// TIA Portal V17 export
// export: Created 2025-03-05T08:01:40.8595336Z, ExportSetting WithDefaults, DisplayName Totally Integrated Automation Portal, DisplayVersion V17 Update 8, DisplayName TIA Portal Openness, DisplayVersion V17 Update 8, DisplayName TIA Portal Version Control Interface, DisplayVersion V17, DisplayName SINAMICS Startdrive Advanced, DisplayVersion V17 SP2, DisplayName SINAMICS Startdrive G110M, G120, G120C, G120D, G120P, G115D, DisplayVersion V17 SP2, DisplayName SINAMICS Startdrive G130, G150, S120, S150, SINAMICS MV, S210, DisplayVersion V17 SP2, DisplayName STEP 7 Professional, DisplayVersion V17 Update 8, DisplayName SINUMERIK ONE STEP 7 Toolbox, DisplayVersion V17 Update 12, DisplayName SINUMERIK 840D sl STEP 7 Toolbox, DisplayVersion V17 Update 12, DisplayName STEP 7 Safety, DisplayVersion V17 Update 6, DisplayName WinCC Advanced, DisplayVersion V17 Update 8
FUNCTION "FC7238_HMI_WINCC_OVERVIEW" : Void   // FC7238, LAD
{ S7_Optimized_Access := 'TRUE' }
VERSION : 0.1
// stored: AutoNumber false, IsIECCheckEnabled false, SetENOAutomatically false, UDAEnableTagReadback false
   VAR_TEMP
      RETVAL_FILL : Int;
   END_VAR
BEGIN

REGION Network 1: UNIT 01 ASPIRATION ALL STATIONS READY
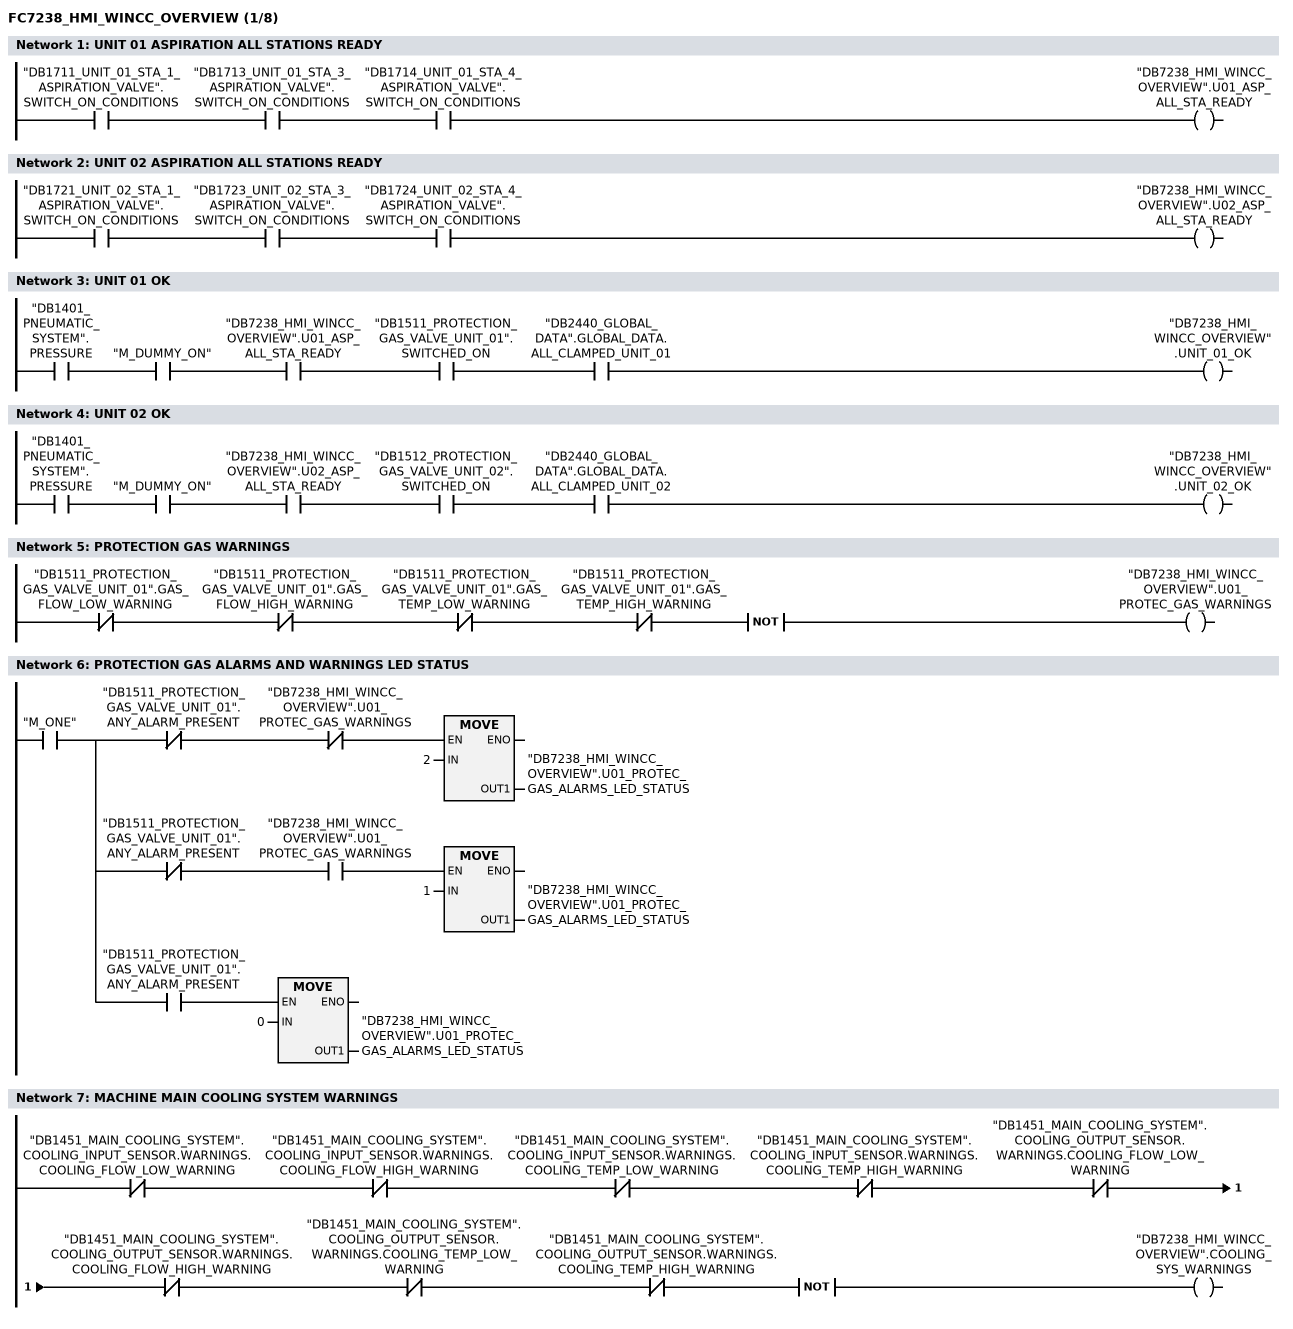
   RUNG wire#powerrail
      Contact( "DB1711_UNIT_01_STA_1_ASPIRATION_VALVE".SWITCH_ON_CONDITIONS )
      Contact( "DB1713_UNIT_01_STA_3_ASPIRATION_VALVE".SWITCH_ON_CONDITIONS )
      Contact( "DB1714_UNIT_01_STA_4_ASPIRATION_VALVE".SWITCH_ON_CONDITIONS )
      Coil( "DB7238_HMI_WINCC_OVERVIEW".U01_ASP_ALL_STA_READY )
   END_RUNG
   // the same network as SCL:
   "DB7238_HMI_WINCC_OVERVIEW".U01_ASP_ALL_STA_READY := "DB1711_UNIT_01_STA_1_ASPIRATION_VALVE".SWITCH_ON_CONDITIONS AND "DB1713_UNIT_01_STA_3_ASPIRATION_VALVE".SWITCH_ON_CONDITIONS AND "DB1714_UNIT_01_STA_4_ASPIRATION_VALVE".SWITCH_ON_CONDITIONS;
END_REGION

REGION Network 2: UNIT 02 ASPIRATION ALL STATIONS READY
   RUNG wire#powerrail
      Contact( "DB1721_UNIT_02_STA_1_ASPIRATION_VALVE".SWITCH_ON_CONDITIONS )
      Contact( "DB1723_UNIT_02_STA_3_ASPIRATION_VALVE".SWITCH_ON_CONDITIONS )
      Contact( "DB1724_UNIT_02_STA_4_ASPIRATION_VALVE".SWITCH_ON_CONDITIONS )
      Coil( "DB7238_HMI_WINCC_OVERVIEW".U02_ASP_ALL_STA_READY )
   END_RUNG
   // the same network as SCL:
   "DB7238_HMI_WINCC_OVERVIEW".U02_ASP_ALL_STA_READY := "DB1721_UNIT_02_STA_1_ASPIRATION_VALVE".SWITCH_ON_CONDITIONS AND "DB1723_UNIT_02_STA_3_ASPIRATION_VALVE".SWITCH_ON_CONDITIONS AND "DB1724_UNIT_02_STA_4_ASPIRATION_VALVE".SWITCH_ON_CONDITIONS;
END_REGION

REGION Network 3: UNIT 01 OK
   RUNG wire#powerrail
      Contact( "DB1401_PNEUMATIC_SYSTEM".PRESSURE )
      Contact( "M_DUMMY_ON" )
      Contact( "DB7238_HMI_WINCC_OVERVIEW".U01_ASP_ALL_STA_READY )
      Contact( "DB1511_PROTECTION_GAS_VALVE_UNIT_01".SWITCHED_ON )
      Contact( "DB2440_GLOBAL_DATA".GLOBAL_DATA.ALL_CLAMPED_UNIT_01 )
      Coil( "DB7238_HMI_WINCC_OVERVIEW".UNIT_01_OK )
   END_RUNG
   // the same network as SCL:
   "DB7238_HMI_WINCC_OVERVIEW".UNIT_01_OK := "DB1401_PNEUMATIC_SYSTEM".PRESSURE AND "M_DUMMY_ON" AND "DB7238_HMI_WINCC_OVERVIEW".U01_ASP_ALL_STA_READY AND "DB1511_PROTECTION_GAS_VALVE_UNIT_01".SWITCHED_ON AND "DB2440_GLOBAL_DATA".GLOBAL_DATA.ALL_CLAMPED_UNIT_01;
END_REGION

REGION Network 4: UNIT 02 OK
   RUNG wire#powerrail
      Contact( "DB1401_PNEUMATIC_SYSTEM".PRESSURE )
      Contact( "M_DUMMY_ON" )
      Contact( "DB7238_HMI_WINCC_OVERVIEW".U02_ASP_ALL_STA_READY )
      Contact( "DB1512_PROTECTION_GAS_VALVE_UNIT_02".SWITCHED_ON )
      Contact( "DB2440_GLOBAL_DATA".GLOBAL_DATA.ALL_CLAMPED_UNIT_02 )
      Coil( "DB7238_HMI_WINCC_OVERVIEW".UNIT_02_OK )
   END_RUNG
   // the same network as SCL:
   "DB7238_HMI_WINCC_OVERVIEW".UNIT_02_OK := "DB1401_PNEUMATIC_SYSTEM".PRESSURE AND "M_DUMMY_ON" AND "DB7238_HMI_WINCC_OVERVIEW".U02_ASP_ALL_STA_READY AND "DB1512_PROTECTION_GAS_VALVE_UNIT_02".SWITCHED_ON AND "DB2440_GLOBAL_DATA".GLOBAL_DATA.ALL_CLAMPED_UNIT_02;
END_REGION

REGION Network 5: PROTECTION GAS WARNINGS
   RUNG wire#powerrail
      I_Contact( "DB1511_PROTECTION_GAS_VALVE_UNIT_01".GAS_FLOW_LOW_WARNING )
      I_Contact( "DB1511_PROTECTION_GAS_VALVE_UNIT_01".GAS_FLOW_HIGH_WARNING )
      I_Contact( "DB1511_PROTECTION_GAS_VALVE_UNIT_01".GAS_TEMP_LOW_WARNING )
      I_Contact( "DB1511_PROTECTION_GAS_VALVE_UNIT_01".GAS_TEMP_HIGH_WARNING )
      Not()
      Coil( "DB7238_HMI_WINCC_OVERVIEW".U01_PROTEC_GAS_WARNINGS )
   END_RUNG
   // the same network as SCL:
   "DB7238_HMI_WINCC_OVERVIEW".U01_PROTEC_GAS_WARNINGS := NOT (NOT "DB1511_PROTECTION_GAS_VALVE_UNIT_01".GAS_FLOW_LOW_WARNING AND NOT "DB1511_PROTECTION_GAS_VALVE_UNIT_01".GAS_FLOW_HIGH_WARNING AND NOT "DB1511_PROTECTION_GAS_VALVE_UNIT_01".GAS_TEMP_LOW_WARNING AND NOT "DB1511_PROTECTION_GAS_VALVE_UNIT_01".GAS_TEMP_HIGH_WARNING);
END_REGION

REGION Network 6: PROTECTION GAS ALARMS AND WARNINGS LED STATUS
   RUNG wire#powerrail
      Contact( "M_ONE" )
      wire#w1
      I_Contact( "DB1511_PROTECTION_GAS_VALVE_UNIT_01".ANY_ALARM_PRESENT )
      I_Contact( "DB7238_HMI_WINCC_OVERVIEW".U01_PROTEC_GAS_WARNINGS )
      { S7_GenerateENO := "TRUE" } Move(in := 2, out1 => "DB7238_HMI_WINCC_OVERVIEW".U01_PROTEC_GAS_ALARMS_LED_STATUS)
   END_RUNG
   RUNG wire#w1
      I_Contact( "DB1511_PROTECTION_GAS_VALVE_UNIT_01".ANY_ALARM_PRESENT )
      Contact( "DB7238_HMI_WINCC_OVERVIEW".U01_PROTEC_GAS_WARNINGS )
      { S7_GenerateENO := "TRUE" } Move(in := 1, out1 => "DB7238_HMI_WINCC_OVERVIEW".U01_PROTEC_GAS_ALARMS_LED_STATUS)
   END_RUNG
   RUNG wire#w1
      Contact( "DB1511_PROTECTION_GAS_VALVE_UNIT_01".ANY_ALARM_PRESENT )
      { S7_GenerateENO := "TRUE" } Move(in := 0, out1 => "DB7238_HMI_WINCC_OVERVIEW".U01_PROTEC_GAS_ALARMS_LED_STATUS)
   END_RUNG
   // the same network as SCL:
   IF "M_ONE" AND NOT "DB1511_PROTECTION_GAS_VALVE_UNIT_01".ANY_ALARM_PRESENT AND NOT "DB7238_HMI_WINCC_OVERVIEW".U01_PROTEC_GAS_WARNINGS THEN
       "DB7238_HMI_WINCC_OVERVIEW".U01_PROTEC_GAS_ALARMS_LED_STATUS := 2;
   END_IF;
   IF "M_ONE" AND NOT "DB1511_PROTECTION_GAS_VALVE_UNIT_01".ANY_ALARM_PRESENT AND "DB7238_HMI_WINCC_OVERVIEW".U01_PROTEC_GAS_WARNINGS THEN
       "DB7238_HMI_WINCC_OVERVIEW".U01_PROTEC_GAS_ALARMS_LED_STATUS := 1;
   END_IF;
   IF "M_ONE" AND "DB1511_PROTECTION_GAS_VALVE_UNIT_01".ANY_ALARM_PRESENT THEN
       "DB7238_HMI_WINCC_OVERVIEW".U01_PROTEC_GAS_ALARMS_LED_STATUS := 0;
   END_IF;
END_REGION

REGION Network 7: MACHINE MAIN COOLING SYSTEM WARNINGS
   RUNG wire#powerrail
      I_Contact( "DB1451_MAIN_COOLING_SYSTEM".COOLING_INPUT_SENSOR.WARNINGS.COOLING_FLOW_LOW_WARNING )
      I_Contact( "DB1451_MAIN_COOLING_SYSTEM".COOLING_INPUT_SENSOR.WARNINGS.COOLING_FLOW_HIGH_WARNING )
      I_Contact( "DB1451_MAIN_COOLING_SYSTEM".COOLING_INPUT_SENSOR.WARNINGS.COOLING_TEMP_LOW_WARNING )
      I_Contact( "DB1451_MAIN_COOLING_SYSTEM".COOLING_INPUT_SENSOR.WARNINGS.COOLING_TEMP_HIGH_WARNING )
      I_Contact( "DB1451_MAIN_COOLING_SYSTEM".COOLING_OUTPUT_SENSOR.WARNINGS.COOLING_FLOW_LOW_WARNING )
      I_Contact( "DB1451_MAIN_COOLING_SYSTEM".COOLING_OUTPUT_SENSOR.WARNINGS.COOLING_FLOW_HIGH_WARNING )
      I_Contact( "DB1451_MAIN_COOLING_SYSTEM".COOLING_OUTPUT_SENSOR.WARNINGS.COOLING_TEMP_LOW_WARNING )
      I_Contact( "DB1451_MAIN_COOLING_SYSTEM".COOLING_OUTPUT_SENSOR.WARNINGS.COOLING_TEMP_HIGH_WARNING )
      Not()
      Coil( "DB7238_HMI_WINCC_OVERVIEW".COOLING_SYS_WARNINGS )
   END_RUNG
   // the same network as SCL:
   "DB7238_HMI_WINCC_OVERVIEW".COOLING_SYS_WARNINGS := NOT (NOT "DB1451_MAIN_COOLING_SYSTEM".COOLING_INPUT_SENSOR.WARNINGS.COOLING_FLOW_LOW_WARNING AND NOT "DB1451_MAIN_COOLING_SYSTEM".COOLING_INPUT_SENSOR.WARNINGS.COOLING_FLOW_HIGH_WARNING AND NOT "DB1451_MAIN_COOLING_SYSTEM".COOLING_INPUT_SENSOR.WARNINGS.COOLING_TEMP_LOW_WARNING AND NOT "DB1451_MAIN_COOLING_SYSTEM".COOLING_INPUT_SENSOR.WARNINGS.COOLING_TEMP_HIGH_WARNING AND NOT "DB1451_MAIN_COOLING_SYSTEM".COOLING_OUTPUT_SENSOR.WARNINGS.COOLING_FLOW_LOW_WARNING AND NOT "DB1451_MAIN_COOLING_SYSTEM".COOLING_OUTPUT_SENSOR.WARNINGS.COOLING_FLOW_HIGH_WARNING AND NOT "DB1451_MAIN_COOLING_SYSTEM".COOLING_OUTPUT_SENSOR.WARNINGS.COOLING_TEMP_LOW_WARNING AND NOT "DB1451_MAIN_COOLING_SYSTEM".COOLING_OUTPUT_SENSOR.WARNINGS.COOLING_TEMP_HIGH_WARNING);
END_REGION

REGION Network 8: MACHINE MAIN COOLING SYSTEM ALARMS
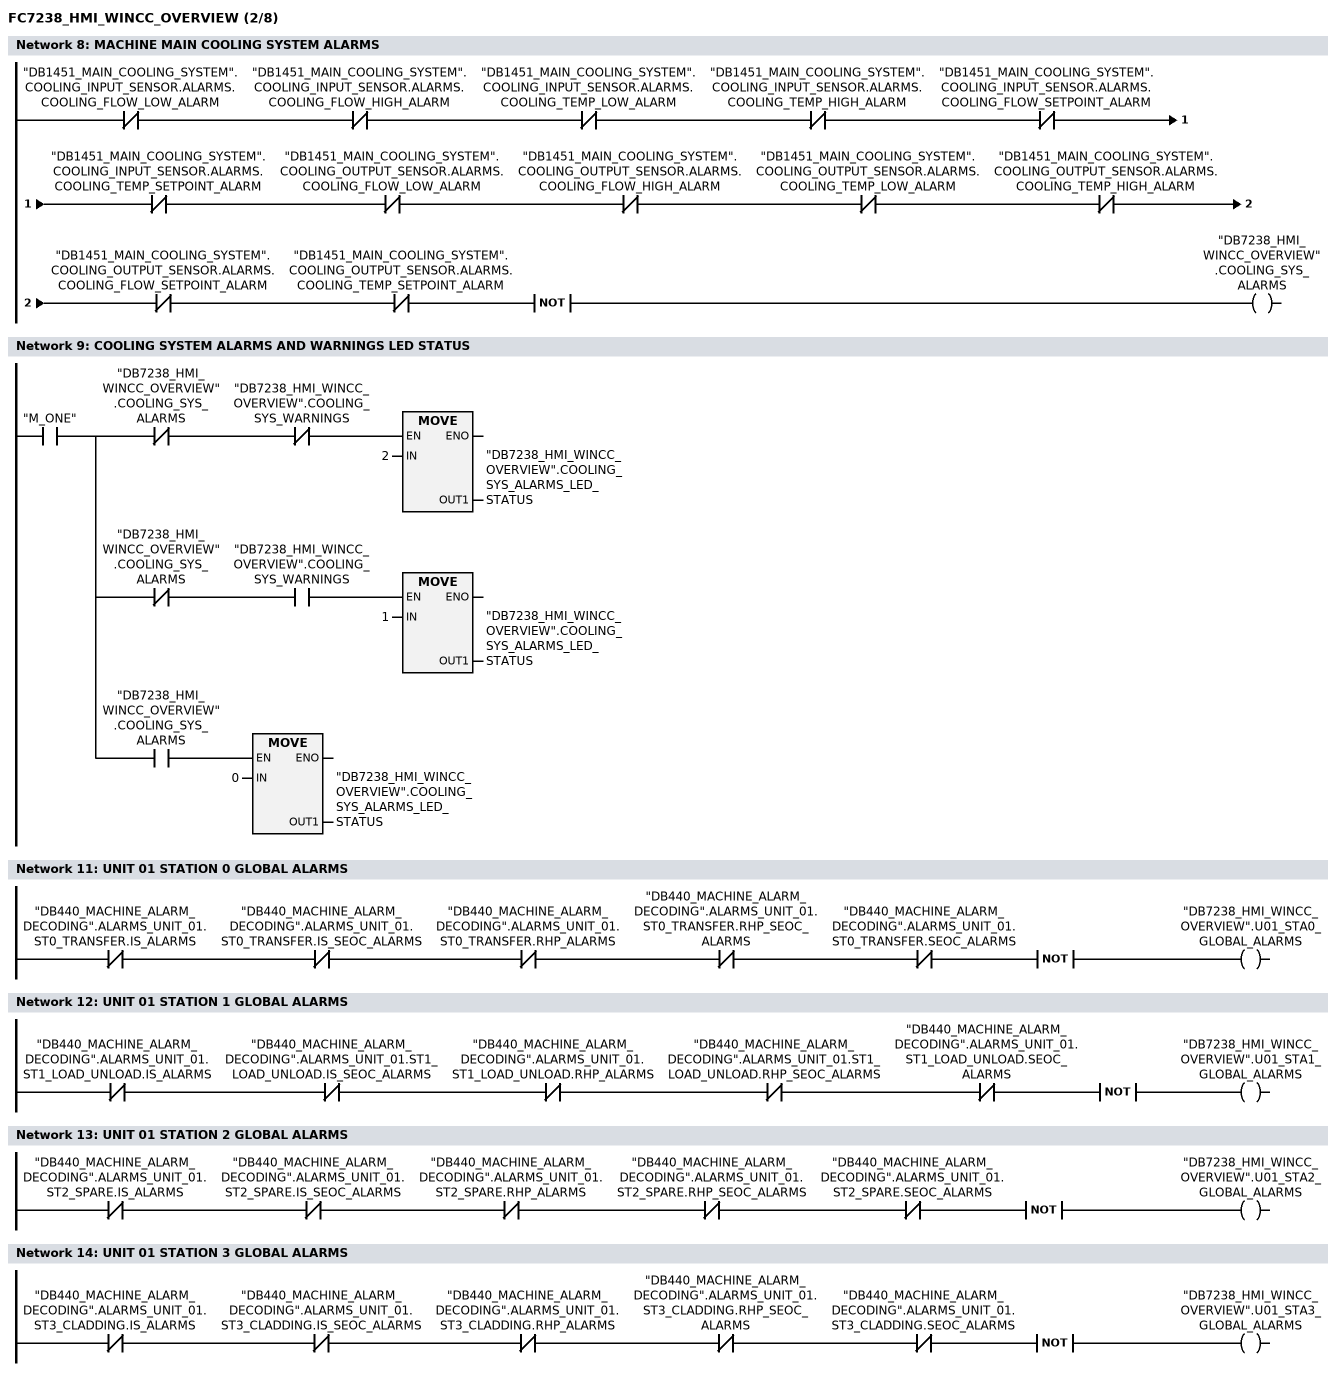
   RUNG wire#powerrail
      I_Contact( "DB1451_MAIN_COOLING_SYSTEM".COOLING_INPUT_SENSOR.ALARMS.COOLING_FLOW_LOW_ALARM )
      I_Contact( "DB1451_MAIN_COOLING_SYSTEM".COOLING_INPUT_SENSOR.ALARMS.COOLING_FLOW_HIGH_ALARM )
      I_Contact( "DB1451_MAIN_COOLING_SYSTEM".COOLING_INPUT_SENSOR.ALARMS.COOLING_TEMP_LOW_ALARM )
      I_Contact( "DB1451_MAIN_COOLING_SYSTEM".COOLING_INPUT_SENSOR.ALARMS.COOLING_TEMP_HIGH_ALARM )
      I_Contact( "DB1451_MAIN_COOLING_SYSTEM".COOLING_INPUT_SENSOR.ALARMS.COOLING_FLOW_SETPOINT_ALARM )
      I_Contact( "DB1451_MAIN_COOLING_SYSTEM".COOLING_INPUT_SENSOR.ALARMS.COOLING_TEMP_SETPOINT_ALARM )
      I_Contact( "DB1451_MAIN_COOLING_SYSTEM".COOLING_OUTPUT_SENSOR.ALARMS.COOLING_FLOW_LOW_ALARM )
      I_Contact( "DB1451_MAIN_COOLING_SYSTEM".COOLING_OUTPUT_SENSOR.ALARMS.COOLING_FLOW_HIGH_ALARM )
      I_Contact( "DB1451_MAIN_COOLING_SYSTEM".COOLING_OUTPUT_SENSOR.ALARMS.COOLING_TEMP_LOW_ALARM )
      I_Contact( "DB1451_MAIN_COOLING_SYSTEM".COOLING_OUTPUT_SENSOR.ALARMS.COOLING_TEMP_HIGH_ALARM )
      I_Contact( "DB1451_MAIN_COOLING_SYSTEM".COOLING_OUTPUT_SENSOR.ALARMS.COOLING_FLOW_SETPOINT_ALARM )
      I_Contact( "DB1451_MAIN_COOLING_SYSTEM".COOLING_OUTPUT_SENSOR.ALARMS.COOLING_TEMP_SETPOINT_ALARM )
      Not()
      Coil( "DB7238_HMI_WINCC_OVERVIEW".COOLING_SYS_ALARMS )
   END_RUNG
   // the same network as SCL:
   "DB7238_HMI_WINCC_OVERVIEW".COOLING_SYS_ALARMS := NOT (NOT "DB1451_MAIN_COOLING_SYSTEM".COOLING_INPUT_SENSOR.ALARMS.COOLING_FLOW_LOW_ALARM AND NOT "DB1451_MAIN_COOLING_SYSTEM".COOLING_INPUT_SENSOR.ALARMS.COOLING_FLOW_HIGH_ALARM AND NOT "DB1451_MAIN_COOLING_SYSTEM".COOLING_INPUT_SENSOR.ALARMS.COOLING_TEMP_LOW_ALARM AND NOT "DB1451_MAIN_COOLING_SYSTEM".COOLING_INPUT_SENSOR.ALARMS.COOLING_TEMP_HIGH_ALARM AND NOT "DB1451_MAIN_COOLING_SYSTEM".COOLING_INPUT_SENSOR.ALARMS.COOLING_FLOW_SETPOINT_ALARM AND NOT "DB1451_MAIN_COOLING_SYSTEM".COOLING_INPUT_SENSOR.ALARMS.COOLING_TEMP_SETPOINT_ALARM AND NOT "DB1451_MAIN_COOLING_SYSTEM".COOLING_OUTPUT_SENSOR.ALARMS.COOLING_FLOW_LOW_ALARM AND NOT "DB1451_MAIN_COOLING_SYSTEM".COOLING_OUTPUT_SENSOR.ALARMS.COOLING_FLOW_HIGH_ALARM AND NOT "DB1451_MAIN_COOLING_SYSTEM".COOLING_OUTPUT_SENSOR.ALARMS.COOLING_TEMP_LOW_ALARM AND NOT "DB1451_MAIN_COOLING_SYSTEM".COOLING_OUTPUT_SENSOR.ALARMS.COOLING_TEMP_HIGH_ALARM AND NOT "DB1451_MAIN_COOLING_SYSTEM".COOLING_OUTPUT_SENSOR.ALARMS.COOLING_FLOW_SETPOINT_ALARM AND NOT "DB1451_MAIN_COOLING_SYSTEM".COOLING_OUTPUT_SENSOR.ALARMS.COOLING_TEMP_SETPOINT_ALARM);
END_REGION

REGION Network 9: COOLING SYSTEM ALARMS AND WARNINGS LED STATUS
   RUNG wire#powerrail
      Contact( "M_ONE" )
      wire#w1
      I_Contact( "DB7238_HMI_WINCC_OVERVIEW".COOLING_SYS_ALARMS )
      I_Contact( "DB7238_HMI_WINCC_OVERVIEW".COOLING_SYS_WARNINGS )
      { S7_GenerateENO := "TRUE" } Move(in := 2, out1 => "DB7238_HMI_WINCC_OVERVIEW".COOLING_SYS_ALARMS_LED_STATUS)
   END_RUNG
   RUNG wire#w1
      I_Contact( "DB7238_HMI_WINCC_OVERVIEW".COOLING_SYS_ALARMS )
      Contact( "DB7238_HMI_WINCC_OVERVIEW".COOLING_SYS_WARNINGS )
      { S7_GenerateENO := "TRUE" } Move(in := 1, out1 => "DB7238_HMI_WINCC_OVERVIEW".COOLING_SYS_ALARMS_LED_STATUS)
   END_RUNG
   RUNG wire#w1
      Contact( "DB7238_HMI_WINCC_OVERVIEW".COOLING_SYS_ALARMS )
      { S7_GenerateENO := "TRUE" } Move(in := 0, out1 => "DB7238_HMI_WINCC_OVERVIEW".COOLING_SYS_ALARMS_LED_STATUS)
   END_RUNG
   // the same network as SCL:
   IF "M_ONE" AND NOT "DB7238_HMI_WINCC_OVERVIEW".COOLING_SYS_ALARMS AND NOT "DB7238_HMI_WINCC_OVERVIEW".COOLING_SYS_WARNINGS THEN
       "DB7238_HMI_WINCC_OVERVIEW".COOLING_SYS_ALARMS_LED_STATUS := 2;
   END_IF;
   IF "M_ONE" AND NOT "DB7238_HMI_WINCC_OVERVIEW".COOLING_SYS_ALARMS AND "DB7238_HMI_WINCC_OVERVIEW".COOLING_SYS_WARNINGS THEN
       "DB7238_HMI_WINCC_OVERVIEW".COOLING_SYS_ALARMS_LED_STATUS := 1;
   END_IF;
   IF "M_ONE" AND "DB7238_HMI_WINCC_OVERVIEW".COOLING_SYS_ALARMS THEN
       "DB7238_HMI_WINCC_OVERVIEW".COOLING_SYS_ALARMS_LED_STATUS := 0;
   END_IF;
END_REGION

REGION Network 10: <<<<<<<<<<<<<<<<<<<<<<<< UNIT 01 >>>>>>>>>>>>>>>>>>>>>>>>
END_REGION

REGION Network 11: UNIT 01 STATION 0 GLOBAL ALARMS
   RUNG wire#powerrail
      I_Contact( "DB440_MACHINE_ALARM_DECODING".ALARMS_UNIT_01.ST0_TRANSFER.IS_ALARMS )
      I_Contact( "DB440_MACHINE_ALARM_DECODING".ALARMS_UNIT_01.ST0_TRANSFER.IS_SEOC_ALARMS )
      I_Contact( "DB440_MACHINE_ALARM_DECODING".ALARMS_UNIT_01.ST0_TRANSFER.RHP_ALARMS )
      I_Contact( "DB440_MACHINE_ALARM_DECODING".ALARMS_UNIT_01.ST0_TRANSFER.RHP_SEOC_ALARMS )
      I_Contact( "DB440_MACHINE_ALARM_DECODING".ALARMS_UNIT_01.ST0_TRANSFER.SEOC_ALARMS )
      Not()
      Coil( "DB7238_HMI_WINCC_OVERVIEW".U01_STA0_GLOBAL_ALARMS )
   END_RUNG
   // the same network as SCL:
   "DB7238_HMI_WINCC_OVERVIEW".U01_STA0_GLOBAL_ALARMS := NOT (NOT "DB440_MACHINE_ALARM_DECODING".ALARMS_UNIT_01.ST0_TRANSFER.IS_ALARMS AND NOT "DB440_MACHINE_ALARM_DECODING".ALARMS_UNIT_01.ST0_TRANSFER.IS_SEOC_ALARMS AND NOT "DB440_MACHINE_ALARM_DECODING".ALARMS_UNIT_01.ST0_TRANSFER.RHP_ALARMS AND NOT "DB440_MACHINE_ALARM_DECODING".ALARMS_UNIT_01.ST0_TRANSFER.RHP_SEOC_ALARMS AND NOT "DB440_MACHINE_ALARM_DECODING".ALARMS_UNIT_01.ST0_TRANSFER.SEOC_ALARMS);
END_REGION

REGION Network 12: UNIT 01 STATION 1 GLOBAL ALARMS
   RUNG wire#powerrail
      I_Contact( "DB440_MACHINE_ALARM_DECODING".ALARMS_UNIT_01.ST1_LOAD_UNLOAD.IS_ALARMS )
      I_Contact( "DB440_MACHINE_ALARM_DECODING".ALARMS_UNIT_01.ST1_LOAD_UNLOAD.IS_SEOC_ALARMS )
      I_Contact( "DB440_MACHINE_ALARM_DECODING".ALARMS_UNIT_01.ST1_LOAD_UNLOAD.RHP_ALARMS )
      I_Contact( "DB440_MACHINE_ALARM_DECODING".ALARMS_UNIT_01.ST1_LOAD_UNLOAD.RHP_SEOC_ALARMS )
      I_Contact( "DB440_MACHINE_ALARM_DECODING".ALARMS_UNIT_01.ST1_LOAD_UNLOAD.SEOC_ALARMS )
      Not()
      Coil( "DB7238_HMI_WINCC_OVERVIEW".U01_STA1_GLOBAL_ALARMS )
   END_RUNG
   // the same network as SCL:
   "DB7238_HMI_WINCC_OVERVIEW".U01_STA1_GLOBAL_ALARMS := NOT (NOT "DB440_MACHINE_ALARM_DECODING".ALARMS_UNIT_01.ST1_LOAD_UNLOAD.IS_ALARMS AND NOT "DB440_MACHINE_ALARM_DECODING".ALARMS_UNIT_01.ST1_LOAD_UNLOAD.IS_SEOC_ALARMS AND NOT "DB440_MACHINE_ALARM_DECODING".ALARMS_UNIT_01.ST1_LOAD_UNLOAD.RHP_ALARMS AND NOT "DB440_MACHINE_ALARM_DECODING".ALARMS_UNIT_01.ST1_LOAD_UNLOAD.RHP_SEOC_ALARMS AND NOT "DB440_MACHINE_ALARM_DECODING".ALARMS_UNIT_01.ST1_LOAD_UNLOAD.SEOC_ALARMS);
END_REGION

REGION Network 13: UNIT 01 STATION 2 GLOBAL ALARMS
   RUNG wire#powerrail
      I_Contact( "DB440_MACHINE_ALARM_DECODING".ALARMS_UNIT_01.ST2_SPARE.IS_ALARMS )
      I_Contact( "DB440_MACHINE_ALARM_DECODING".ALARMS_UNIT_01.ST2_SPARE.IS_SEOC_ALARMS )
      I_Contact( "DB440_MACHINE_ALARM_DECODING".ALARMS_UNIT_01.ST2_SPARE.RHP_ALARMS )
      I_Contact( "DB440_MACHINE_ALARM_DECODING".ALARMS_UNIT_01.ST2_SPARE.RHP_SEOC_ALARMS )
      I_Contact( "DB440_MACHINE_ALARM_DECODING".ALARMS_UNIT_01.ST2_SPARE.SEOC_ALARMS )
      Not()
      Coil( "DB7238_HMI_WINCC_OVERVIEW".U01_STA2_GLOBAL_ALARMS )
   END_RUNG
   // the same network as SCL:
   "DB7238_HMI_WINCC_OVERVIEW".U01_STA2_GLOBAL_ALARMS := NOT (NOT "DB440_MACHINE_ALARM_DECODING".ALARMS_UNIT_01.ST2_SPARE.IS_ALARMS AND NOT "DB440_MACHINE_ALARM_DECODING".ALARMS_UNIT_01.ST2_SPARE.IS_SEOC_ALARMS AND NOT "DB440_MACHINE_ALARM_DECODING".ALARMS_UNIT_01.ST2_SPARE.RHP_ALARMS AND NOT "DB440_MACHINE_ALARM_DECODING".ALARMS_UNIT_01.ST2_SPARE.RHP_SEOC_ALARMS AND NOT "DB440_MACHINE_ALARM_DECODING".ALARMS_UNIT_01.ST2_SPARE.SEOC_ALARMS);
END_REGION

REGION Network 14: UNIT 01 STATION 3 GLOBAL ALARMS
   RUNG wire#powerrail
      I_Contact( "DB440_MACHINE_ALARM_DECODING".ALARMS_UNIT_01.ST3_CLADDING.IS_ALARMS )
      I_Contact( "DB440_MACHINE_ALARM_DECODING".ALARMS_UNIT_01.ST3_CLADDING.IS_SEOC_ALARMS )
      I_Contact( "DB440_MACHINE_ALARM_DECODING".ALARMS_UNIT_01.ST3_CLADDING.RHP_ALARMS )
      I_Contact( "DB440_MACHINE_ALARM_DECODING".ALARMS_UNIT_01.ST3_CLADDING.RHP_SEOC_ALARMS )
      I_Contact( "DB440_MACHINE_ALARM_DECODING".ALARMS_UNIT_01.ST3_CLADDING.SEOC_ALARMS )
      Not()
      Coil( "DB7238_HMI_WINCC_OVERVIEW".U01_STA3_GLOBAL_ALARMS )
   END_RUNG
   // the same network as SCL:
   "DB7238_HMI_WINCC_OVERVIEW".U01_STA3_GLOBAL_ALARMS := NOT (NOT "DB440_MACHINE_ALARM_DECODING".ALARMS_UNIT_01.ST3_CLADDING.IS_ALARMS AND NOT "DB440_MACHINE_ALARM_DECODING".ALARMS_UNIT_01.ST3_CLADDING.IS_SEOC_ALARMS AND NOT "DB440_MACHINE_ALARM_DECODING".ALARMS_UNIT_01.ST3_CLADDING.RHP_ALARMS AND NOT "DB440_MACHINE_ALARM_DECODING".ALARMS_UNIT_01.ST3_CLADDING.RHP_SEOC_ALARMS AND NOT "DB440_MACHINE_ALARM_DECODING".ALARMS_UNIT_01.ST3_CLADDING.SEOC_ALARMS);
END_REGION

REGION Network 15: UNIT 01 STATION 4 GLOBAL ALARMS
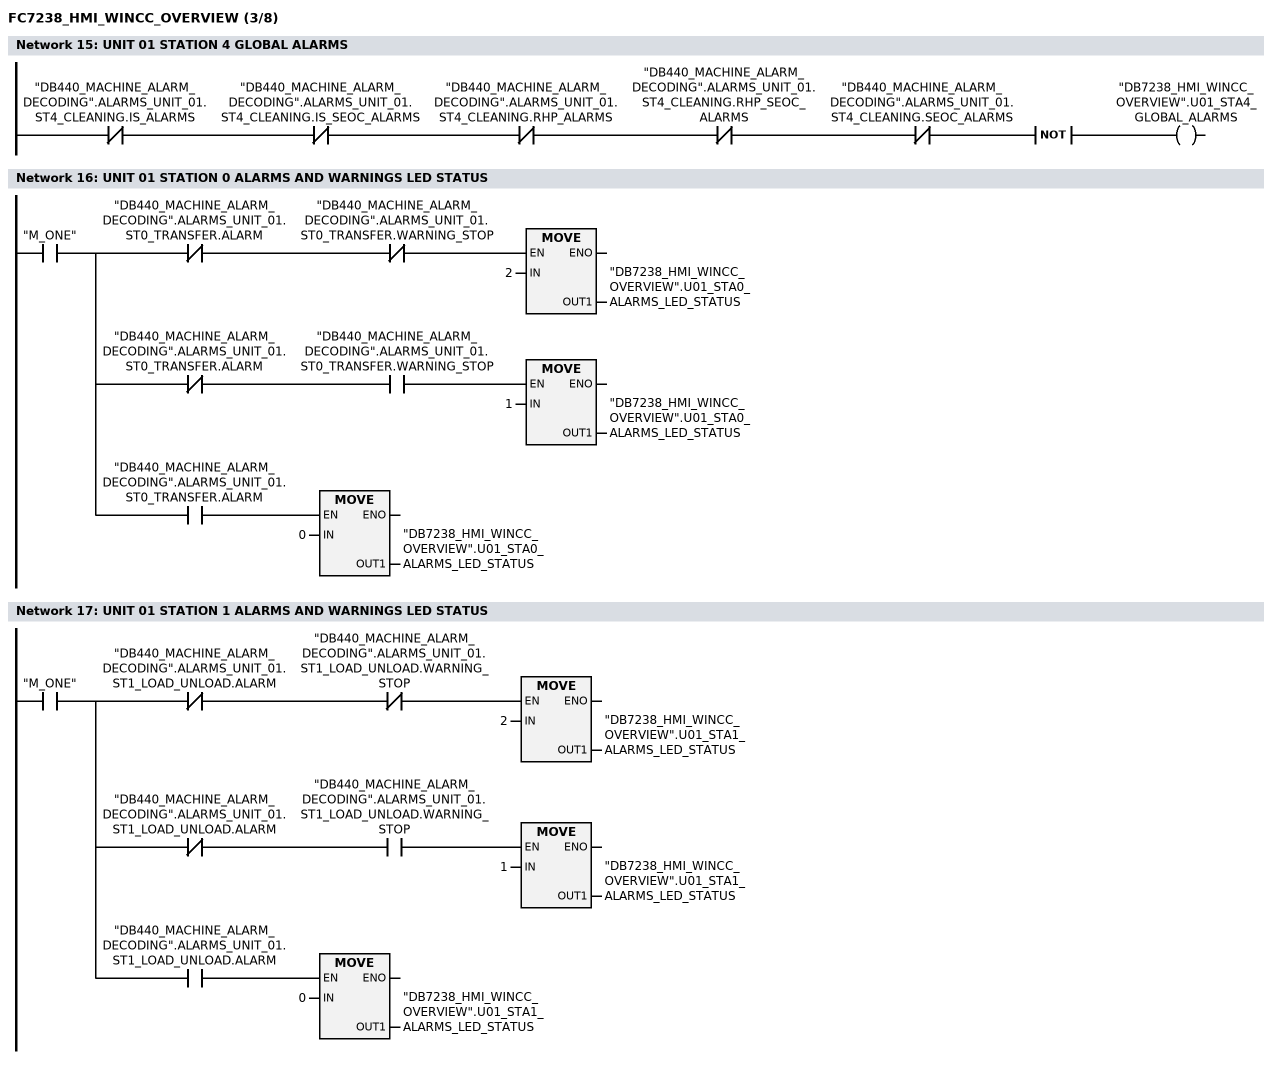
   RUNG wire#powerrail
      I_Contact( "DB440_MACHINE_ALARM_DECODING".ALARMS_UNIT_01.ST4_CLEANING.IS_ALARMS )
      I_Contact( "DB440_MACHINE_ALARM_DECODING".ALARMS_UNIT_01.ST4_CLEANING.IS_SEOC_ALARMS )
      I_Contact( "DB440_MACHINE_ALARM_DECODING".ALARMS_UNIT_01.ST4_CLEANING.RHP_ALARMS )
      I_Contact( "DB440_MACHINE_ALARM_DECODING".ALARMS_UNIT_01.ST4_CLEANING.RHP_SEOC_ALARMS )
      I_Contact( "DB440_MACHINE_ALARM_DECODING".ALARMS_UNIT_01.ST4_CLEANING.SEOC_ALARMS )
      Not()
      Coil( "DB7238_HMI_WINCC_OVERVIEW".U01_STA4_GLOBAL_ALARMS )
   END_RUNG
   // the same network as SCL:
   "DB7238_HMI_WINCC_OVERVIEW".U01_STA4_GLOBAL_ALARMS := NOT (NOT "DB440_MACHINE_ALARM_DECODING".ALARMS_UNIT_01.ST4_CLEANING.IS_ALARMS AND NOT "DB440_MACHINE_ALARM_DECODING".ALARMS_UNIT_01.ST4_CLEANING.IS_SEOC_ALARMS AND NOT "DB440_MACHINE_ALARM_DECODING".ALARMS_UNIT_01.ST4_CLEANING.RHP_ALARMS AND NOT "DB440_MACHINE_ALARM_DECODING".ALARMS_UNIT_01.ST4_CLEANING.RHP_SEOC_ALARMS AND NOT "DB440_MACHINE_ALARM_DECODING".ALARMS_UNIT_01.ST4_CLEANING.SEOC_ALARMS);
END_REGION

REGION Network 16: UNIT 01 STATION 0 ALARMS AND WARNINGS LED STATUS
   RUNG wire#powerrail
      Contact( "M_ONE" )
      wire#w1
      I_Contact( "DB440_MACHINE_ALARM_DECODING".ALARMS_UNIT_01.ST0_TRANSFER.ALARM )
      I_Contact( "DB440_MACHINE_ALARM_DECODING".ALARMS_UNIT_01.ST0_TRANSFER.WARNING_STOP )
      { S7_GenerateENO := "TRUE" } Move(in := 2, out1 => "DB7238_HMI_WINCC_OVERVIEW".U01_STA0_ALARMS_LED_STATUS)
   END_RUNG
   RUNG wire#w1
      I_Contact( "DB440_MACHINE_ALARM_DECODING".ALARMS_UNIT_01.ST0_TRANSFER.ALARM )
      Contact( "DB440_MACHINE_ALARM_DECODING".ALARMS_UNIT_01.ST0_TRANSFER.WARNING_STOP )
      { S7_GenerateENO := "TRUE" } Move(in := 1, out1 => "DB7238_HMI_WINCC_OVERVIEW".U01_STA0_ALARMS_LED_STATUS)
   END_RUNG
   RUNG wire#w1
      Contact( "DB440_MACHINE_ALARM_DECODING".ALARMS_UNIT_01.ST0_TRANSFER.ALARM )
      { S7_GenerateENO := "TRUE" } Move(in := 0, out1 => "DB7238_HMI_WINCC_OVERVIEW".U01_STA0_ALARMS_LED_STATUS)
   END_RUNG
   // the same network as SCL:
   IF "M_ONE" AND NOT "DB440_MACHINE_ALARM_DECODING".ALARMS_UNIT_01.ST0_TRANSFER.ALARM AND NOT "DB440_MACHINE_ALARM_DECODING".ALARMS_UNIT_01.ST0_TRANSFER.WARNING_STOP THEN
       "DB7238_HMI_WINCC_OVERVIEW".U01_STA0_ALARMS_LED_STATUS := 2;
   END_IF;
   IF "M_ONE" AND NOT "DB440_MACHINE_ALARM_DECODING".ALARMS_UNIT_01.ST0_TRANSFER.ALARM AND "DB440_MACHINE_ALARM_DECODING".ALARMS_UNIT_01.ST0_TRANSFER.WARNING_STOP THEN
       "DB7238_HMI_WINCC_OVERVIEW".U01_STA0_ALARMS_LED_STATUS := 1;
   END_IF;
   IF "M_ONE" AND "DB440_MACHINE_ALARM_DECODING".ALARMS_UNIT_01.ST0_TRANSFER.ALARM THEN
       "DB7238_HMI_WINCC_OVERVIEW".U01_STA0_ALARMS_LED_STATUS := 0;
   END_IF;
END_REGION

REGION Network 17: UNIT 01 STATION 1 ALARMS AND WARNINGS LED STATUS
   RUNG wire#powerrail
      Contact( "M_ONE" )
      wire#w1
      I_Contact( "DB440_MACHINE_ALARM_DECODING".ALARMS_UNIT_01.ST1_LOAD_UNLOAD.ALARM )
      I_Contact( "DB440_MACHINE_ALARM_DECODING".ALARMS_UNIT_01.ST1_LOAD_UNLOAD.WARNING_STOP )
      { S7_GenerateENO := "TRUE" } Move(in := 2, out1 => "DB7238_HMI_WINCC_OVERVIEW".U01_STA1_ALARMS_LED_STATUS)
   END_RUNG
   RUNG wire#w1
      I_Contact( "DB440_MACHINE_ALARM_DECODING".ALARMS_UNIT_01.ST1_LOAD_UNLOAD.ALARM )
      Contact( "DB440_MACHINE_ALARM_DECODING".ALARMS_UNIT_01.ST1_LOAD_UNLOAD.WARNING_STOP )
      { S7_GenerateENO := "TRUE" } Move(in := 1, out1 => "DB7238_HMI_WINCC_OVERVIEW".U01_STA1_ALARMS_LED_STATUS)
   END_RUNG
   RUNG wire#w1
      Contact( "DB440_MACHINE_ALARM_DECODING".ALARMS_UNIT_01.ST1_LOAD_UNLOAD.ALARM )
      { S7_GenerateENO := "TRUE" } Move(in := 0, out1 => "DB7238_HMI_WINCC_OVERVIEW".U01_STA1_ALARMS_LED_STATUS)
   END_RUNG
   // the same network as SCL:
   IF "M_ONE" AND NOT "DB440_MACHINE_ALARM_DECODING".ALARMS_UNIT_01.ST1_LOAD_UNLOAD.ALARM AND NOT "DB440_MACHINE_ALARM_DECODING".ALARMS_UNIT_01.ST1_LOAD_UNLOAD.WARNING_STOP THEN
       "DB7238_HMI_WINCC_OVERVIEW".U01_STA1_ALARMS_LED_STATUS := 2;
   END_IF;
   IF "M_ONE" AND NOT "DB440_MACHINE_ALARM_DECODING".ALARMS_UNIT_01.ST1_LOAD_UNLOAD.ALARM AND "DB440_MACHINE_ALARM_DECODING".ALARMS_UNIT_01.ST1_LOAD_UNLOAD.WARNING_STOP THEN
       "DB7238_HMI_WINCC_OVERVIEW".U01_STA1_ALARMS_LED_STATUS := 1;
   END_IF;
   IF "M_ONE" AND "DB440_MACHINE_ALARM_DECODING".ALARMS_UNIT_01.ST1_LOAD_UNLOAD.ALARM THEN
       "DB7238_HMI_WINCC_OVERVIEW".U01_STA1_ALARMS_LED_STATUS := 0;
   END_IF;
END_REGION

REGION Network 18: UNIT 01 STATION 2 ALARMS AND WARNINGS LED STATUS
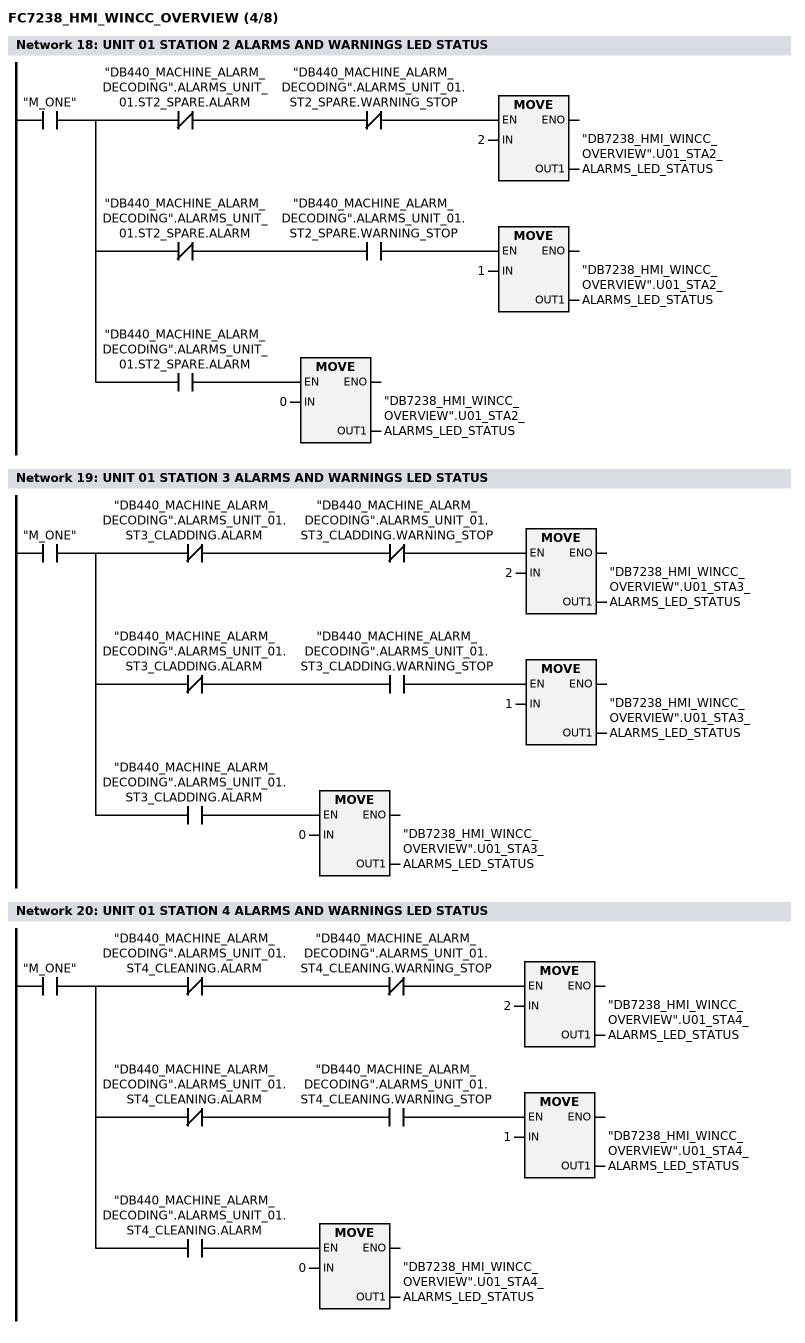
   RUNG wire#powerrail
      Contact( "M_ONE" )
      wire#w1
      I_Contact( "DB440_MACHINE_ALARM_DECODING".ALARMS_UNIT_01.ST2_SPARE.ALARM )
      I_Contact( "DB440_MACHINE_ALARM_DECODING".ALARMS_UNIT_01.ST2_SPARE.WARNING_STOP )
      { S7_GenerateENO := "TRUE" } Move(in := 2, out1 => "DB7238_HMI_WINCC_OVERVIEW".U01_STA2_ALARMS_LED_STATUS)
   END_RUNG
   RUNG wire#w1
      I_Contact( "DB440_MACHINE_ALARM_DECODING".ALARMS_UNIT_01.ST2_SPARE.ALARM )
      Contact( "DB440_MACHINE_ALARM_DECODING".ALARMS_UNIT_01.ST2_SPARE.WARNING_STOP )
      { S7_GenerateENO := "TRUE" } Move(in := 1, out1 => "DB7238_HMI_WINCC_OVERVIEW".U01_STA2_ALARMS_LED_STATUS)
   END_RUNG
   RUNG wire#w1
      Contact( "DB440_MACHINE_ALARM_DECODING".ALARMS_UNIT_01.ST2_SPARE.ALARM )
      { S7_GenerateENO := "TRUE" } Move(in := 0, out1 => "DB7238_HMI_WINCC_OVERVIEW".U01_STA2_ALARMS_LED_STATUS)
   END_RUNG
   // the same network as SCL:
   IF "M_ONE" AND NOT "DB440_MACHINE_ALARM_DECODING".ALARMS_UNIT_01.ST2_SPARE.ALARM AND NOT "DB440_MACHINE_ALARM_DECODING".ALARMS_UNIT_01.ST2_SPARE.WARNING_STOP THEN
       "DB7238_HMI_WINCC_OVERVIEW".U01_STA2_ALARMS_LED_STATUS := 2;
   END_IF;
   IF "M_ONE" AND NOT "DB440_MACHINE_ALARM_DECODING".ALARMS_UNIT_01.ST2_SPARE.ALARM AND "DB440_MACHINE_ALARM_DECODING".ALARMS_UNIT_01.ST2_SPARE.WARNING_STOP THEN
       "DB7238_HMI_WINCC_OVERVIEW".U01_STA2_ALARMS_LED_STATUS := 1;
   END_IF;
   IF "M_ONE" AND "DB440_MACHINE_ALARM_DECODING".ALARMS_UNIT_01.ST2_SPARE.ALARM THEN
       "DB7238_HMI_WINCC_OVERVIEW".U01_STA2_ALARMS_LED_STATUS := 0;
   END_IF;
END_REGION

REGION Network 19: UNIT 01 STATION 3 ALARMS AND WARNINGS LED STATUS
   RUNG wire#powerrail
      Contact( "M_ONE" )
      wire#w1
      I_Contact( "DB440_MACHINE_ALARM_DECODING".ALARMS_UNIT_01.ST3_CLADDING.ALARM )
      I_Contact( "DB440_MACHINE_ALARM_DECODING".ALARMS_UNIT_01.ST3_CLADDING.WARNING_STOP )
      { S7_GenerateENO := "TRUE" } Move(in := 2, out1 => "DB7238_HMI_WINCC_OVERVIEW".U01_STA3_ALARMS_LED_STATUS)
   END_RUNG
   RUNG wire#w1
      I_Contact( "DB440_MACHINE_ALARM_DECODING".ALARMS_UNIT_01.ST3_CLADDING.ALARM )
      Contact( "DB440_MACHINE_ALARM_DECODING".ALARMS_UNIT_01.ST3_CLADDING.WARNING_STOP )
      { S7_GenerateENO := "TRUE" } Move(in := 1, out1 => "DB7238_HMI_WINCC_OVERVIEW".U01_STA3_ALARMS_LED_STATUS)
   END_RUNG
   RUNG wire#w1
      Contact( "DB440_MACHINE_ALARM_DECODING".ALARMS_UNIT_01.ST3_CLADDING.ALARM )
      { S7_GenerateENO := "TRUE" } Move(in := 0, out1 => "DB7238_HMI_WINCC_OVERVIEW".U01_STA3_ALARMS_LED_STATUS)
   END_RUNG
   // the same network as SCL:
   IF "M_ONE" AND NOT "DB440_MACHINE_ALARM_DECODING".ALARMS_UNIT_01.ST3_CLADDING.ALARM AND NOT "DB440_MACHINE_ALARM_DECODING".ALARMS_UNIT_01.ST3_CLADDING.WARNING_STOP THEN
       "DB7238_HMI_WINCC_OVERVIEW".U01_STA3_ALARMS_LED_STATUS := 2;
   END_IF;
   IF "M_ONE" AND NOT "DB440_MACHINE_ALARM_DECODING".ALARMS_UNIT_01.ST3_CLADDING.ALARM AND "DB440_MACHINE_ALARM_DECODING".ALARMS_UNIT_01.ST3_CLADDING.WARNING_STOP THEN
       "DB7238_HMI_WINCC_OVERVIEW".U01_STA3_ALARMS_LED_STATUS := 1;
   END_IF;
   IF "M_ONE" AND "DB440_MACHINE_ALARM_DECODING".ALARMS_UNIT_01.ST3_CLADDING.ALARM THEN
       "DB7238_HMI_WINCC_OVERVIEW".U01_STA3_ALARMS_LED_STATUS := 0;
   END_IF;
END_REGION

REGION Network 20: UNIT 01 STATION 4 ALARMS AND WARNINGS LED STATUS
   RUNG wire#powerrail
      Contact( "M_ONE" )
      wire#w1
      I_Contact( "DB440_MACHINE_ALARM_DECODING".ALARMS_UNIT_01.ST4_CLEANING.ALARM )
      I_Contact( "DB440_MACHINE_ALARM_DECODING".ALARMS_UNIT_01.ST4_CLEANING.WARNING_STOP )
      { S7_GenerateENO := "TRUE" } Move(in := 2, out1 => "DB7238_HMI_WINCC_OVERVIEW".U01_STA4_ALARMS_LED_STATUS)
   END_RUNG
   RUNG wire#w1
      I_Contact( "DB440_MACHINE_ALARM_DECODING".ALARMS_UNIT_01.ST4_CLEANING.ALARM )
      Contact( "DB440_MACHINE_ALARM_DECODING".ALARMS_UNIT_01.ST4_CLEANING.WARNING_STOP )
      { S7_GenerateENO := "TRUE" } Move(in := 1, out1 => "DB7238_HMI_WINCC_OVERVIEW".U01_STA4_ALARMS_LED_STATUS)
   END_RUNG
   RUNG wire#w1
      Contact( "DB440_MACHINE_ALARM_DECODING".ALARMS_UNIT_01.ST4_CLEANING.ALARM )
      { S7_GenerateENO := "TRUE" } Move(in := 0, out1 => "DB7238_HMI_WINCC_OVERVIEW".U01_STA4_ALARMS_LED_STATUS)
   END_RUNG
   // the same network as SCL:
   IF "M_ONE" AND NOT "DB440_MACHINE_ALARM_DECODING".ALARMS_UNIT_01.ST4_CLEANING.ALARM AND NOT "DB440_MACHINE_ALARM_DECODING".ALARMS_UNIT_01.ST4_CLEANING.WARNING_STOP THEN
       "DB7238_HMI_WINCC_OVERVIEW".U01_STA4_ALARMS_LED_STATUS := 2;
   END_IF;
   IF "M_ONE" AND NOT "DB440_MACHINE_ALARM_DECODING".ALARMS_UNIT_01.ST4_CLEANING.ALARM AND "DB440_MACHINE_ALARM_DECODING".ALARMS_UNIT_01.ST4_CLEANING.WARNING_STOP THEN
       "DB7238_HMI_WINCC_OVERVIEW".U01_STA4_ALARMS_LED_STATUS := 1;
   END_IF;
   IF "M_ONE" AND "DB440_MACHINE_ALARM_DECODING".ALARMS_UNIT_01.ST4_CLEANING.ALARM THEN
       "DB7238_HMI_WINCC_OVERVIEW".U01_STA4_ALARMS_LED_STATUS := 0;
   END_IF;
END_REGION

REGION Network 21: UNIT 01 ALL FIXTURES CLAMP ALARMS
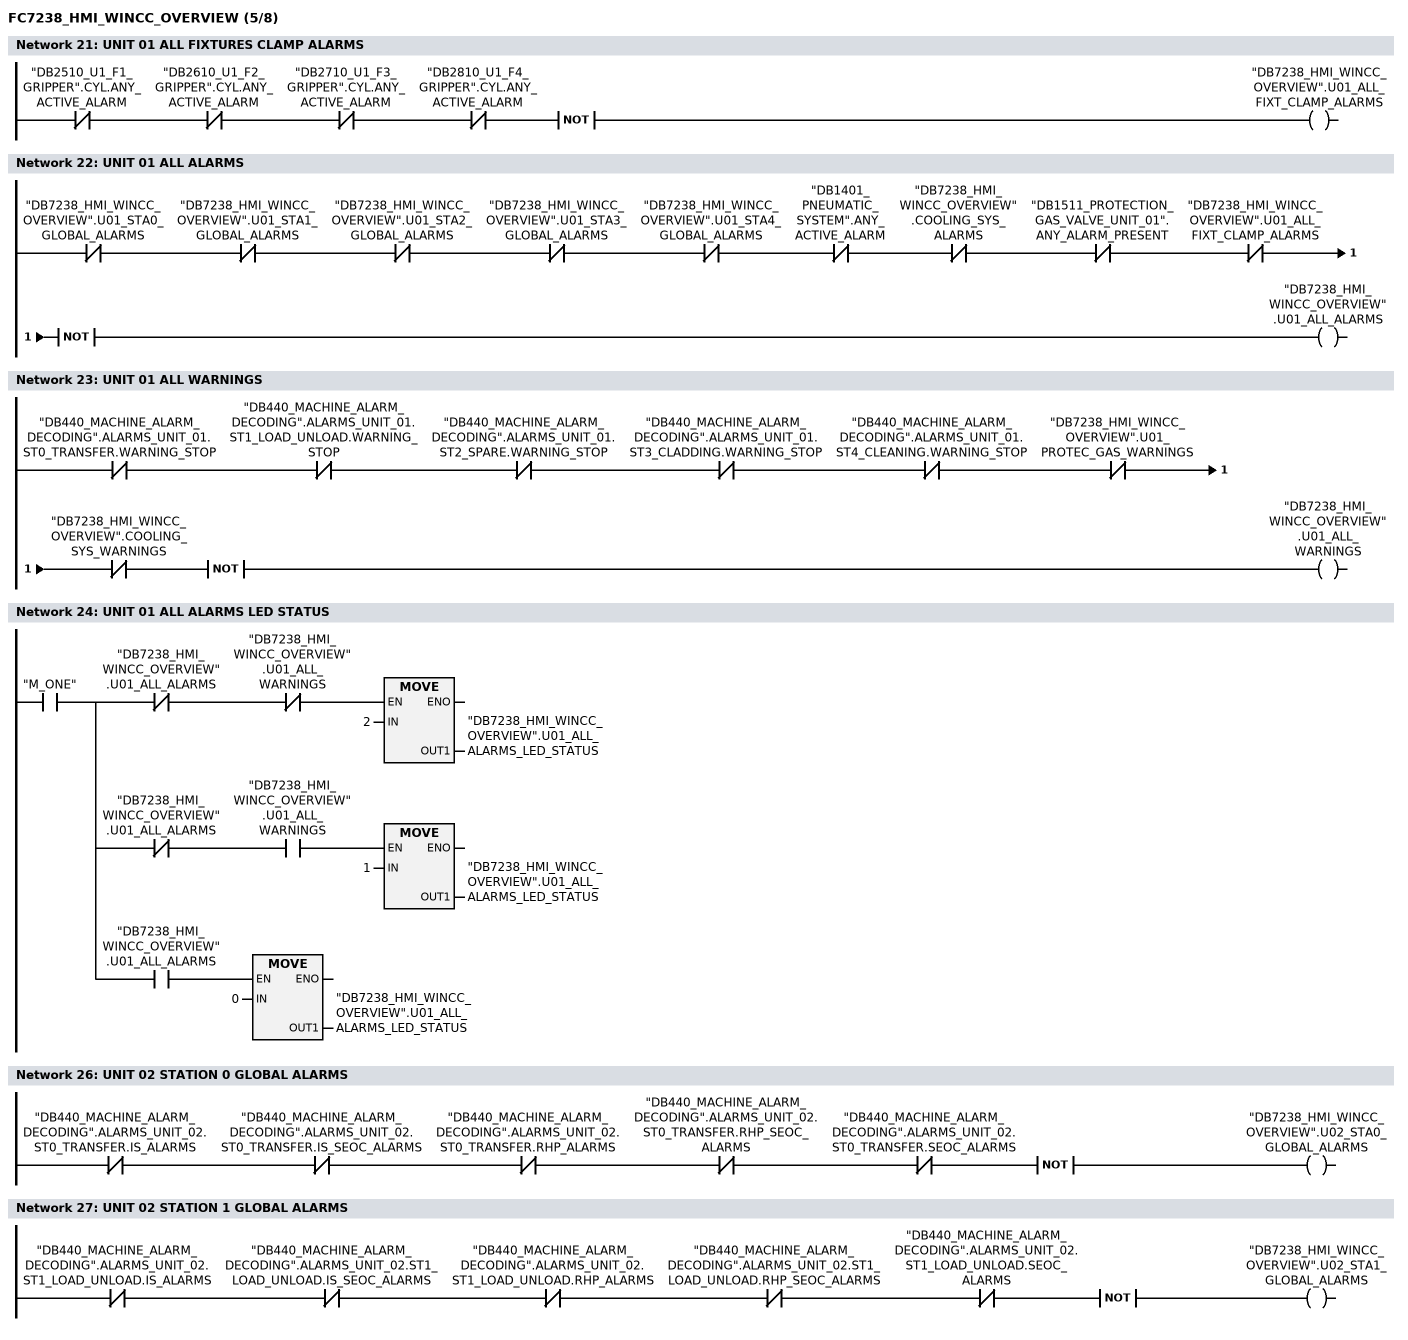
   RUNG wire#powerrail
      I_Contact( "DB2510_U1_F1_GRIPPER".CYL.ANY_ACTIVE_ALARM )
      I_Contact( "DB2610_U1_F2_GRIPPER".CYL.ANY_ACTIVE_ALARM )
      I_Contact( "DB2710_U1_F3_GRIPPER".CYL.ANY_ACTIVE_ALARM )
      I_Contact( "DB2810_U1_F4_GRIPPER".CYL.ANY_ACTIVE_ALARM )
      Not()
      Coil( "DB7238_HMI_WINCC_OVERVIEW".U01_ALL_FIXT_CLAMP_ALARMS )
   END_RUNG
   // the same network as SCL:
   "DB7238_HMI_WINCC_OVERVIEW".U01_ALL_FIXT_CLAMP_ALARMS := NOT (NOT "DB2510_U1_F1_GRIPPER".CYL.ANY_ACTIVE_ALARM AND NOT "DB2610_U1_F2_GRIPPER".CYL.ANY_ACTIVE_ALARM AND NOT "DB2710_U1_F3_GRIPPER".CYL.ANY_ACTIVE_ALARM AND NOT "DB2810_U1_F4_GRIPPER".CYL.ANY_ACTIVE_ALARM);
END_REGION

REGION Network 22: UNIT 01 ALL ALARMS
   RUNG wire#powerrail
      I_Contact( "DB7238_HMI_WINCC_OVERVIEW".U01_STA0_GLOBAL_ALARMS )
      I_Contact( "DB7238_HMI_WINCC_OVERVIEW".U01_STA1_GLOBAL_ALARMS )
      I_Contact( "DB7238_HMI_WINCC_OVERVIEW".U01_STA2_GLOBAL_ALARMS )
      I_Contact( "DB7238_HMI_WINCC_OVERVIEW".U01_STA3_GLOBAL_ALARMS )
      I_Contact( "DB7238_HMI_WINCC_OVERVIEW".U01_STA4_GLOBAL_ALARMS )
      I_Contact( "DB1401_PNEUMATIC_SYSTEM".ANY_ACTIVE_ALARM )
      I_Contact( "DB7238_HMI_WINCC_OVERVIEW".COOLING_SYS_ALARMS )
      I_Contact( "DB1511_PROTECTION_GAS_VALVE_UNIT_01".ANY_ALARM_PRESENT )
      I_Contact( "DB7238_HMI_WINCC_OVERVIEW".U01_ALL_FIXT_CLAMP_ALARMS )
      Not()
      Coil( "DB7238_HMI_WINCC_OVERVIEW".U01_ALL_ALARMS )
   END_RUNG
   // the same network as SCL:
   "DB7238_HMI_WINCC_OVERVIEW".U01_ALL_ALARMS := NOT (NOT "DB7238_HMI_WINCC_OVERVIEW".U01_STA0_GLOBAL_ALARMS AND NOT "DB7238_HMI_WINCC_OVERVIEW".U01_STA1_GLOBAL_ALARMS AND NOT "DB7238_HMI_WINCC_OVERVIEW".U01_STA2_GLOBAL_ALARMS AND NOT "DB7238_HMI_WINCC_OVERVIEW".U01_STA3_GLOBAL_ALARMS AND NOT "DB7238_HMI_WINCC_OVERVIEW".U01_STA4_GLOBAL_ALARMS AND NOT "DB1401_PNEUMATIC_SYSTEM".ANY_ACTIVE_ALARM AND NOT "DB7238_HMI_WINCC_OVERVIEW".COOLING_SYS_ALARMS AND NOT "DB1511_PROTECTION_GAS_VALVE_UNIT_01".ANY_ALARM_PRESENT AND NOT "DB7238_HMI_WINCC_OVERVIEW".U01_ALL_FIXT_CLAMP_ALARMS);
END_REGION

REGION Network 23: UNIT 01 ALL WARNINGS
   RUNG wire#powerrail
      I_Contact( "DB440_MACHINE_ALARM_DECODING".ALARMS_UNIT_01.ST0_TRANSFER.WARNING_STOP )
      I_Contact( "DB440_MACHINE_ALARM_DECODING".ALARMS_UNIT_01.ST1_LOAD_UNLOAD.WARNING_STOP )
      I_Contact( "DB440_MACHINE_ALARM_DECODING".ALARMS_UNIT_01.ST2_SPARE.WARNING_STOP )
      I_Contact( "DB440_MACHINE_ALARM_DECODING".ALARMS_UNIT_01.ST3_CLADDING.WARNING_STOP )
      I_Contact( "DB440_MACHINE_ALARM_DECODING".ALARMS_UNIT_01.ST4_CLEANING.WARNING_STOP )
      I_Contact( "DB7238_HMI_WINCC_OVERVIEW".U01_PROTEC_GAS_WARNINGS )
      I_Contact( "DB7238_HMI_WINCC_OVERVIEW".COOLING_SYS_WARNINGS )
      Not()
      Coil( "DB7238_HMI_WINCC_OVERVIEW".U01_ALL_WARNINGS )
   END_RUNG
   // the same network as SCL:
   "DB7238_HMI_WINCC_OVERVIEW".U01_ALL_WARNINGS := NOT (NOT "DB440_MACHINE_ALARM_DECODING".ALARMS_UNIT_01.ST0_TRANSFER.WARNING_STOP AND NOT "DB440_MACHINE_ALARM_DECODING".ALARMS_UNIT_01.ST1_LOAD_UNLOAD.WARNING_STOP AND NOT "DB440_MACHINE_ALARM_DECODING".ALARMS_UNIT_01.ST2_SPARE.WARNING_STOP AND NOT "DB440_MACHINE_ALARM_DECODING".ALARMS_UNIT_01.ST3_CLADDING.WARNING_STOP AND NOT "DB440_MACHINE_ALARM_DECODING".ALARMS_UNIT_01.ST4_CLEANING.WARNING_STOP AND NOT "DB7238_HMI_WINCC_OVERVIEW".U01_PROTEC_GAS_WARNINGS AND NOT "DB7238_HMI_WINCC_OVERVIEW".COOLING_SYS_WARNINGS);
END_REGION

REGION Network 24: UNIT 01 ALL ALARMS LED STATUS
   RUNG wire#powerrail
      Contact( "M_ONE" )
      wire#w1
      I_Contact( "DB7238_HMI_WINCC_OVERVIEW".U01_ALL_ALARMS )
      I_Contact( "DB7238_HMI_WINCC_OVERVIEW".U01_ALL_WARNINGS )
      { S7_GenerateENO := "TRUE" } Move(in := 2, out1 => "DB7238_HMI_WINCC_OVERVIEW".U01_ALL_ALARMS_LED_STATUS)
   END_RUNG
   RUNG wire#w1
      I_Contact( "DB7238_HMI_WINCC_OVERVIEW".U01_ALL_ALARMS )
      Contact( "DB7238_HMI_WINCC_OVERVIEW".U01_ALL_WARNINGS )
      { S7_GenerateENO := "TRUE" } Move(in := 1, out1 => "DB7238_HMI_WINCC_OVERVIEW".U01_ALL_ALARMS_LED_STATUS)
   END_RUNG
   RUNG wire#w1
      Contact( "DB7238_HMI_WINCC_OVERVIEW".U01_ALL_ALARMS )
      { S7_GenerateENO := "TRUE" } Move(in := 0, out1 => "DB7238_HMI_WINCC_OVERVIEW".U01_ALL_ALARMS_LED_STATUS)
   END_RUNG
   // the same network as SCL:
   IF "M_ONE" AND NOT "DB7238_HMI_WINCC_OVERVIEW".U01_ALL_ALARMS AND NOT "DB7238_HMI_WINCC_OVERVIEW".U01_ALL_WARNINGS THEN
       "DB7238_HMI_WINCC_OVERVIEW".U01_ALL_ALARMS_LED_STATUS := 2;
   END_IF;
   IF "M_ONE" AND NOT "DB7238_HMI_WINCC_OVERVIEW".U01_ALL_ALARMS AND "DB7238_HMI_WINCC_OVERVIEW".U01_ALL_WARNINGS THEN
       "DB7238_HMI_WINCC_OVERVIEW".U01_ALL_ALARMS_LED_STATUS := 1;
   END_IF;
   IF "M_ONE" AND "DB7238_HMI_WINCC_OVERVIEW".U01_ALL_ALARMS THEN
       "DB7238_HMI_WINCC_OVERVIEW".U01_ALL_ALARMS_LED_STATUS := 0;
   END_IF;
END_REGION

REGION Network 25: <<<<<<<<<<<<<<<<<<<<<<<< UNIT 02 >>>>>>>>>>>>>>>>>>>>>>>>
END_REGION

REGION Network 26: UNIT 02 STATION 0 GLOBAL ALARMS
   RUNG wire#powerrail
      I_Contact( "DB440_MACHINE_ALARM_DECODING".ALARMS_UNIT_02.ST0_TRANSFER.IS_ALARMS )
      I_Contact( "DB440_MACHINE_ALARM_DECODING".ALARMS_UNIT_02.ST0_TRANSFER.IS_SEOC_ALARMS )
      I_Contact( "DB440_MACHINE_ALARM_DECODING".ALARMS_UNIT_02.ST0_TRANSFER.RHP_ALARMS )
      I_Contact( "DB440_MACHINE_ALARM_DECODING".ALARMS_UNIT_02.ST0_TRANSFER.RHP_SEOC_ALARMS )
      I_Contact( "DB440_MACHINE_ALARM_DECODING".ALARMS_UNIT_02.ST0_TRANSFER.SEOC_ALARMS )
      Not()
      Coil( "DB7238_HMI_WINCC_OVERVIEW".U02_STA0_GLOBAL_ALARMS )
   END_RUNG
   // the same network as SCL:
   "DB7238_HMI_WINCC_OVERVIEW".U02_STA0_GLOBAL_ALARMS := NOT (NOT "DB440_MACHINE_ALARM_DECODING".ALARMS_UNIT_02.ST0_TRANSFER.IS_ALARMS AND NOT "DB440_MACHINE_ALARM_DECODING".ALARMS_UNIT_02.ST0_TRANSFER.IS_SEOC_ALARMS AND NOT "DB440_MACHINE_ALARM_DECODING".ALARMS_UNIT_02.ST0_TRANSFER.RHP_ALARMS AND NOT "DB440_MACHINE_ALARM_DECODING".ALARMS_UNIT_02.ST0_TRANSFER.RHP_SEOC_ALARMS AND NOT "DB440_MACHINE_ALARM_DECODING".ALARMS_UNIT_02.ST0_TRANSFER.SEOC_ALARMS);
END_REGION

REGION Network 27: UNIT 02 STATION 1 GLOBAL ALARMS
   RUNG wire#powerrail
      I_Contact( "DB440_MACHINE_ALARM_DECODING".ALARMS_UNIT_02.ST1_LOAD_UNLOAD.IS_ALARMS )
      I_Contact( "DB440_MACHINE_ALARM_DECODING".ALARMS_UNIT_02.ST1_LOAD_UNLOAD.IS_SEOC_ALARMS )
      I_Contact( "DB440_MACHINE_ALARM_DECODING".ALARMS_UNIT_02.ST1_LOAD_UNLOAD.RHP_ALARMS )
      I_Contact( "DB440_MACHINE_ALARM_DECODING".ALARMS_UNIT_02.ST1_LOAD_UNLOAD.RHP_SEOC_ALARMS )
      I_Contact( "DB440_MACHINE_ALARM_DECODING".ALARMS_UNIT_02.ST1_LOAD_UNLOAD.SEOC_ALARMS )
      Not()
      Coil( "DB7238_HMI_WINCC_OVERVIEW".U02_STA1_GLOBAL_ALARMS )
   END_RUNG
   // the same network as SCL:
   "DB7238_HMI_WINCC_OVERVIEW".U02_STA1_GLOBAL_ALARMS := NOT (NOT "DB440_MACHINE_ALARM_DECODING".ALARMS_UNIT_02.ST1_LOAD_UNLOAD.IS_ALARMS AND NOT "DB440_MACHINE_ALARM_DECODING".ALARMS_UNIT_02.ST1_LOAD_UNLOAD.IS_SEOC_ALARMS AND NOT "DB440_MACHINE_ALARM_DECODING".ALARMS_UNIT_02.ST1_LOAD_UNLOAD.RHP_ALARMS AND NOT "DB440_MACHINE_ALARM_DECODING".ALARMS_UNIT_02.ST1_LOAD_UNLOAD.RHP_SEOC_ALARMS AND NOT "DB440_MACHINE_ALARM_DECODING".ALARMS_UNIT_02.ST1_LOAD_UNLOAD.SEOC_ALARMS);
END_REGION

REGION Network 28: UNIT 02 STATION 2 GLOBAL ALARMS
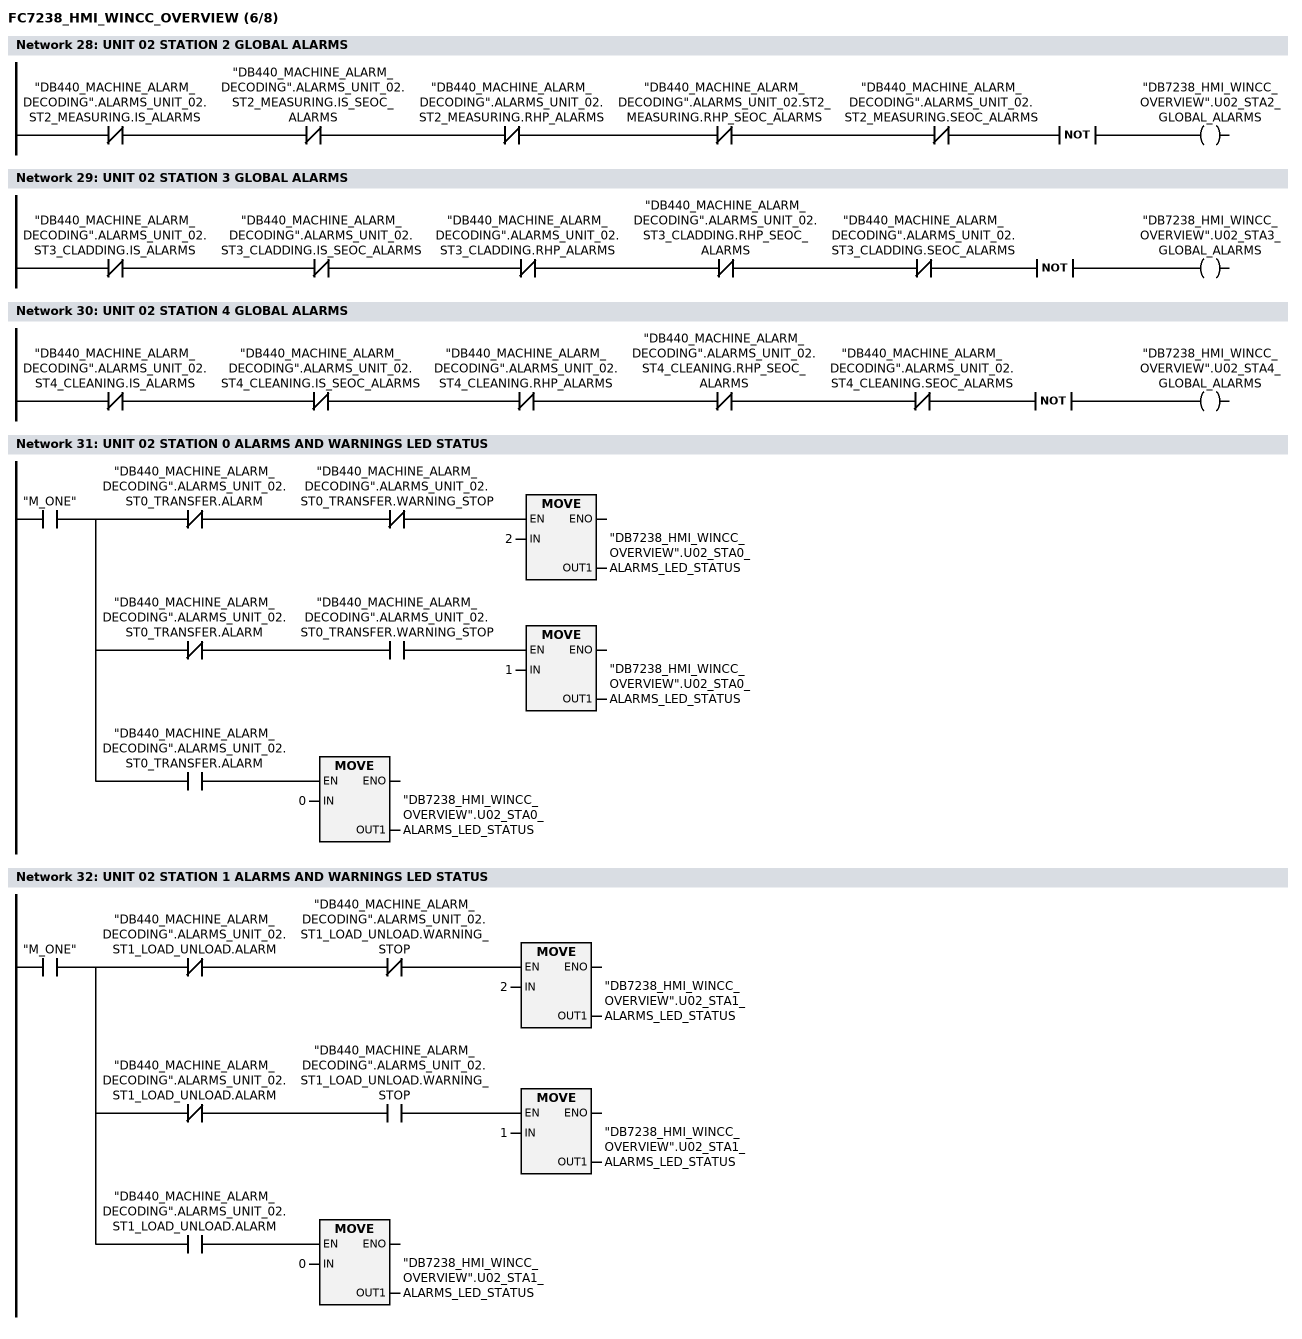
   RUNG wire#powerrail
      I_Contact( "DB440_MACHINE_ALARM_DECODING".ALARMS_UNIT_02.ST2_MEASURING.IS_ALARMS )
      I_Contact( "DB440_MACHINE_ALARM_DECODING".ALARMS_UNIT_02.ST2_MEASURING.IS_SEOC_ALARMS )
      I_Contact( "DB440_MACHINE_ALARM_DECODING".ALARMS_UNIT_02.ST2_MEASURING.RHP_ALARMS )
      I_Contact( "DB440_MACHINE_ALARM_DECODING".ALARMS_UNIT_02.ST2_MEASURING.RHP_SEOC_ALARMS )
      I_Contact( "DB440_MACHINE_ALARM_DECODING".ALARMS_UNIT_02.ST2_MEASURING.SEOC_ALARMS )
      Not()
      Coil( "DB7238_HMI_WINCC_OVERVIEW".U02_STA2_GLOBAL_ALARMS )
   END_RUNG
   // the same network as SCL:
   "DB7238_HMI_WINCC_OVERVIEW".U02_STA2_GLOBAL_ALARMS := NOT (NOT "DB440_MACHINE_ALARM_DECODING".ALARMS_UNIT_02.ST2_MEASURING.IS_ALARMS AND NOT "DB440_MACHINE_ALARM_DECODING".ALARMS_UNIT_02.ST2_MEASURING.IS_SEOC_ALARMS AND NOT "DB440_MACHINE_ALARM_DECODING".ALARMS_UNIT_02.ST2_MEASURING.RHP_ALARMS AND NOT "DB440_MACHINE_ALARM_DECODING".ALARMS_UNIT_02.ST2_MEASURING.RHP_SEOC_ALARMS AND NOT "DB440_MACHINE_ALARM_DECODING".ALARMS_UNIT_02.ST2_MEASURING.SEOC_ALARMS);
END_REGION

REGION Network 29: UNIT 02 STATION 3 GLOBAL ALARMS
   RUNG wire#powerrail
      I_Contact( "DB440_MACHINE_ALARM_DECODING".ALARMS_UNIT_02.ST3_CLADDING.IS_ALARMS )
      I_Contact( "DB440_MACHINE_ALARM_DECODING".ALARMS_UNIT_02.ST3_CLADDING.IS_SEOC_ALARMS )
      I_Contact( "DB440_MACHINE_ALARM_DECODING".ALARMS_UNIT_02.ST3_CLADDING.RHP_ALARMS )
      I_Contact( "DB440_MACHINE_ALARM_DECODING".ALARMS_UNIT_02.ST3_CLADDING.RHP_SEOC_ALARMS )
      I_Contact( "DB440_MACHINE_ALARM_DECODING".ALARMS_UNIT_02.ST3_CLADDING.SEOC_ALARMS )
      Not()
      Coil( "DB7238_HMI_WINCC_OVERVIEW".U02_STA3_GLOBAL_ALARMS )
   END_RUNG
   // the same network as SCL:
   "DB7238_HMI_WINCC_OVERVIEW".U02_STA3_GLOBAL_ALARMS := NOT (NOT "DB440_MACHINE_ALARM_DECODING".ALARMS_UNIT_02.ST3_CLADDING.IS_ALARMS AND NOT "DB440_MACHINE_ALARM_DECODING".ALARMS_UNIT_02.ST3_CLADDING.IS_SEOC_ALARMS AND NOT "DB440_MACHINE_ALARM_DECODING".ALARMS_UNIT_02.ST3_CLADDING.RHP_ALARMS AND NOT "DB440_MACHINE_ALARM_DECODING".ALARMS_UNIT_02.ST3_CLADDING.RHP_SEOC_ALARMS AND NOT "DB440_MACHINE_ALARM_DECODING".ALARMS_UNIT_02.ST3_CLADDING.SEOC_ALARMS);
END_REGION

REGION Network 30: UNIT 02 STATION 4 GLOBAL ALARMS
   RUNG wire#powerrail
      I_Contact( "DB440_MACHINE_ALARM_DECODING".ALARMS_UNIT_02.ST4_CLEANING.IS_ALARMS )
      I_Contact( "DB440_MACHINE_ALARM_DECODING".ALARMS_UNIT_02.ST4_CLEANING.IS_SEOC_ALARMS )
      I_Contact( "DB440_MACHINE_ALARM_DECODING".ALARMS_UNIT_02.ST4_CLEANING.RHP_ALARMS )
      I_Contact( "DB440_MACHINE_ALARM_DECODING".ALARMS_UNIT_02.ST4_CLEANING.RHP_SEOC_ALARMS )
      I_Contact( "DB440_MACHINE_ALARM_DECODING".ALARMS_UNIT_02.ST4_CLEANING.SEOC_ALARMS )
      Not()
      Coil( "DB7238_HMI_WINCC_OVERVIEW".U02_STA4_GLOBAL_ALARMS )
   END_RUNG
   // the same network as SCL:
   "DB7238_HMI_WINCC_OVERVIEW".U02_STA4_GLOBAL_ALARMS := NOT (NOT "DB440_MACHINE_ALARM_DECODING".ALARMS_UNIT_02.ST4_CLEANING.IS_ALARMS AND NOT "DB440_MACHINE_ALARM_DECODING".ALARMS_UNIT_02.ST4_CLEANING.IS_SEOC_ALARMS AND NOT "DB440_MACHINE_ALARM_DECODING".ALARMS_UNIT_02.ST4_CLEANING.RHP_ALARMS AND NOT "DB440_MACHINE_ALARM_DECODING".ALARMS_UNIT_02.ST4_CLEANING.RHP_SEOC_ALARMS AND NOT "DB440_MACHINE_ALARM_DECODING".ALARMS_UNIT_02.ST4_CLEANING.SEOC_ALARMS);
END_REGION

REGION Network 31: UNIT 02 STATION 0 ALARMS AND WARNINGS LED STATUS
   RUNG wire#powerrail
      Contact( "M_ONE" )
      wire#w1
      I_Contact( "DB440_MACHINE_ALARM_DECODING".ALARMS_UNIT_02.ST0_TRANSFER.ALARM )
      I_Contact( "DB440_MACHINE_ALARM_DECODING".ALARMS_UNIT_02.ST0_TRANSFER.WARNING_STOP )
      { S7_GenerateENO := "TRUE" } Move(in := 2, out1 => "DB7238_HMI_WINCC_OVERVIEW".U02_STA0_ALARMS_LED_STATUS)
   END_RUNG
   RUNG wire#w1
      I_Contact( "DB440_MACHINE_ALARM_DECODING".ALARMS_UNIT_02.ST0_TRANSFER.ALARM )
      Contact( "DB440_MACHINE_ALARM_DECODING".ALARMS_UNIT_02.ST0_TRANSFER.WARNING_STOP )
      { S7_GenerateENO := "TRUE" } Move(in := 1, out1 => "DB7238_HMI_WINCC_OVERVIEW".U02_STA0_ALARMS_LED_STATUS)
   END_RUNG
   RUNG wire#w1
      Contact( "DB440_MACHINE_ALARM_DECODING".ALARMS_UNIT_02.ST0_TRANSFER.ALARM )
      { S7_GenerateENO := "TRUE" } Move(in := 0, out1 => "DB7238_HMI_WINCC_OVERVIEW".U02_STA0_ALARMS_LED_STATUS)
   END_RUNG
   // the same network as SCL:
   IF "M_ONE" AND NOT "DB440_MACHINE_ALARM_DECODING".ALARMS_UNIT_02.ST0_TRANSFER.ALARM AND NOT "DB440_MACHINE_ALARM_DECODING".ALARMS_UNIT_02.ST0_TRANSFER.WARNING_STOP THEN
       "DB7238_HMI_WINCC_OVERVIEW".U02_STA0_ALARMS_LED_STATUS := 2;
   END_IF;
   IF "M_ONE" AND NOT "DB440_MACHINE_ALARM_DECODING".ALARMS_UNIT_02.ST0_TRANSFER.ALARM AND "DB440_MACHINE_ALARM_DECODING".ALARMS_UNIT_02.ST0_TRANSFER.WARNING_STOP THEN
       "DB7238_HMI_WINCC_OVERVIEW".U02_STA0_ALARMS_LED_STATUS := 1;
   END_IF;
   IF "M_ONE" AND "DB440_MACHINE_ALARM_DECODING".ALARMS_UNIT_02.ST0_TRANSFER.ALARM THEN
       "DB7238_HMI_WINCC_OVERVIEW".U02_STA0_ALARMS_LED_STATUS := 0;
   END_IF;
END_REGION

REGION Network 32: UNIT 02 STATION 1 ALARMS AND WARNINGS LED STATUS
   RUNG wire#powerrail
      Contact( "M_ONE" )
      wire#w1
      I_Contact( "DB440_MACHINE_ALARM_DECODING".ALARMS_UNIT_02.ST1_LOAD_UNLOAD.ALARM )
      I_Contact( "DB440_MACHINE_ALARM_DECODING".ALARMS_UNIT_02.ST1_LOAD_UNLOAD.WARNING_STOP )
      { S7_GenerateENO := "TRUE" } Move(in := 2, out1 => "DB7238_HMI_WINCC_OVERVIEW".U02_STA1_ALARMS_LED_STATUS)
   END_RUNG
   RUNG wire#w1
      I_Contact( "DB440_MACHINE_ALARM_DECODING".ALARMS_UNIT_02.ST1_LOAD_UNLOAD.ALARM )
      Contact( "DB440_MACHINE_ALARM_DECODING".ALARMS_UNIT_02.ST1_LOAD_UNLOAD.WARNING_STOP )
      { S7_GenerateENO := "TRUE" } Move(in := 1, out1 => "DB7238_HMI_WINCC_OVERVIEW".U02_STA1_ALARMS_LED_STATUS)
   END_RUNG
   RUNG wire#w1
      Contact( "DB440_MACHINE_ALARM_DECODING".ALARMS_UNIT_02.ST1_LOAD_UNLOAD.ALARM )
      { S7_GenerateENO := "TRUE" } Move(in := 0, out1 => "DB7238_HMI_WINCC_OVERVIEW".U02_STA1_ALARMS_LED_STATUS)
   END_RUNG
   // the same network as SCL:
   IF "M_ONE" AND NOT "DB440_MACHINE_ALARM_DECODING".ALARMS_UNIT_02.ST1_LOAD_UNLOAD.ALARM AND NOT "DB440_MACHINE_ALARM_DECODING".ALARMS_UNIT_02.ST1_LOAD_UNLOAD.WARNING_STOP THEN
       "DB7238_HMI_WINCC_OVERVIEW".U02_STA1_ALARMS_LED_STATUS := 2;
   END_IF;
   IF "M_ONE" AND NOT "DB440_MACHINE_ALARM_DECODING".ALARMS_UNIT_02.ST1_LOAD_UNLOAD.ALARM AND "DB440_MACHINE_ALARM_DECODING".ALARMS_UNIT_02.ST1_LOAD_UNLOAD.WARNING_STOP THEN
       "DB7238_HMI_WINCC_OVERVIEW".U02_STA1_ALARMS_LED_STATUS := 1;
   END_IF;
   IF "M_ONE" AND "DB440_MACHINE_ALARM_DECODING".ALARMS_UNIT_02.ST1_LOAD_UNLOAD.ALARM THEN
       "DB7238_HMI_WINCC_OVERVIEW".U02_STA1_ALARMS_LED_STATUS := 0;
   END_IF;
END_REGION

REGION Network 33: UNIT 02 STATION 2 ALARMS AND WARNINGS LED STATUS
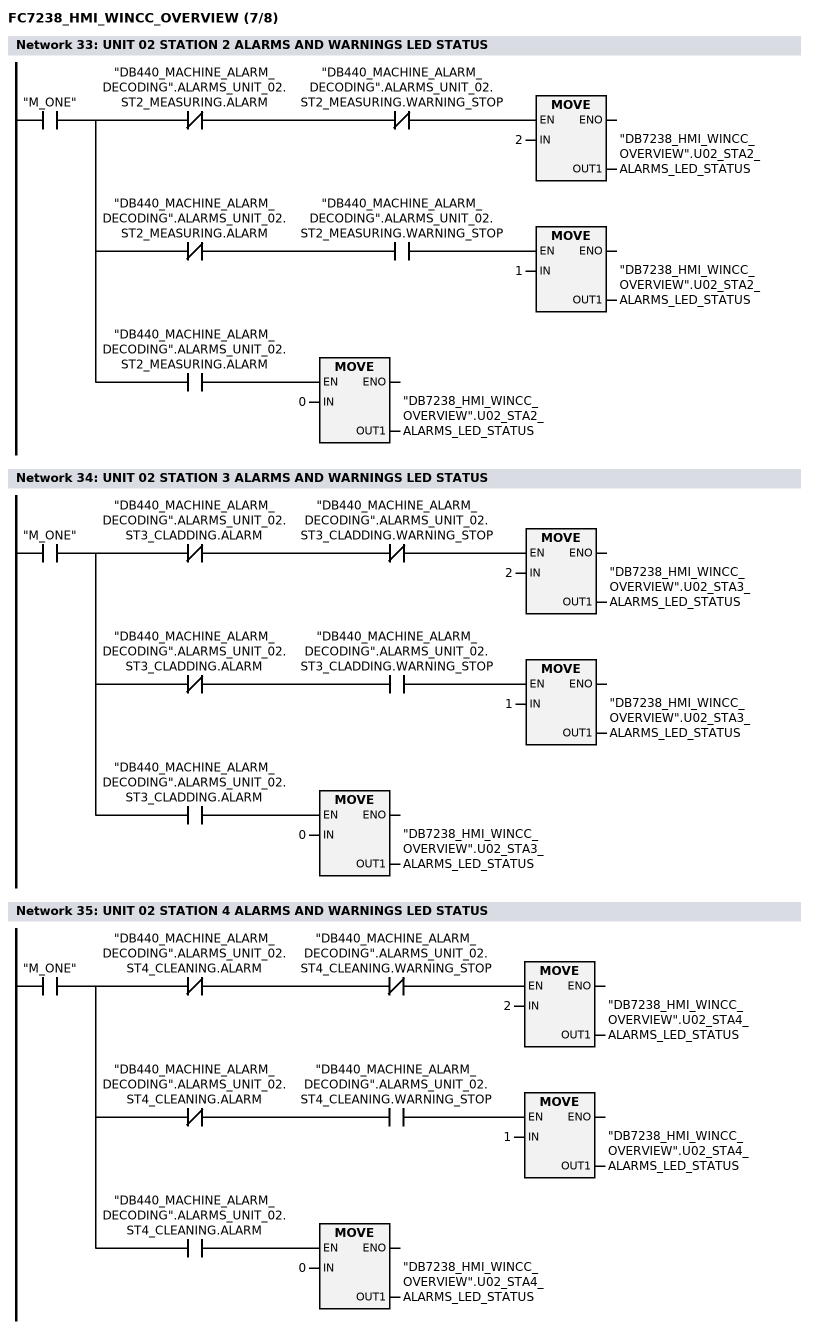
   RUNG wire#powerrail
      Contact( "M_ONE" )
      wire#w1
      I_Contact( "DB440_MACHINE_ALARM_DECODING".ALARMS_UNIT_02.ST2_MEASURING.ALARM )
      I_Contact( "DB440_MACHINE_ALARM_DECODING".ALARMS_UNIT_02.ST2_MEASURING.WARNING_STOP )
      { S7_GenerateENO := "TRUE" } Move(in := 2, out1 => "DB7238_HMI_WINCC_OVERVIEW".U02_STA2_ALARMS_LED_STATUS)
   END_RUNG
   RUNG wire#w1
      I_Contact( "DB440_MACHINE_ALARM_DECODING".ALARMS_UNIT_02.ST2_MEASURING.ALARM )
      Contact( "DB440_MACHINE_ALARM_DECODING".ALARMS_UNIT_02.ST2_MEASURING.WARNING_STOP )
      { S7_GenerateENO := "TRUE" } Move(in := 1, out1 => "DB7238_HMI_WINCC_OVERVIEW".U02_STA2_ALARMS_LED_STATUS)
   END_RUNG
   RUNG wire#w1
      Contact( "DB440_MACHINE_ALARM_DECODING".ALARMS_UNIT_02.ST2_MEASURING.ALARM )
      { S7_GenerateENO := "TRUE" } Move(in := 0, out1 => "DB7238_HMI_WINCC_OVERVIEW".U02_STA2_ALARMS_LED_STATUS)
   END_RUNG
   // the same network as SCL:
   IF "M_ONE" AND NOT "DB440_MACHINE_ALARM_DECODING".ALARMS_UNIT_02.ST2_MEASURING.ALARM AND NOT "DB440_MACHINE_ALARM_DECODING".ALARMS_UNIT_02.ST2_MEASURING.WARNING_STOP THEN
       "DB7238_HMI_WINCC_OVERVIEW".U02_STA2_ALARMS_LED_STATUS := 2;
   END_IF;
   IF "M_ONE" AND NOT "DB440_MACHINE_ALARM_DECODING".ALARMS_UNIT_02.ST2_MEASURING.ALARM AND "DB440_MACHINE_ALARM_DECODING".ALARMS_UNIT_02.ST2_MEASURING.WARNING_STOP THEN
       "DB7238_HMI_WINCC_OVERVIEW".U02_STA2_ALARMS_LED_STATUS := 1;
   END_IF;
   IF "M_ONE" AND "DB440_MACHINE_ALARM_DECODING".ALARMS_UNIT_02.ST2_MEASURING.ALARM THEN
       "DB7238_HMI_WINCC_OVERVIEW".U02_STA2_ALARMS_LED_STATUS := 0;
   END_IF;
END_REGION

REGION Network 34: UNIT 02 STATION 3 ALARMS AND WARNINGS LED STATUS
   RUNG wire#powerrail
      Contact( "M_ONE" )
      wire#w1
      I_Contact( "DB440_MACHINE_ALARM_DECODING".ALARMS_UNIT_02.ST3_CLADDING.ALARM )
      I_Contact( "DB440_MACHINE_ALARM_DECODING".ALARMS_UNIT_02.ST3_CLADDING.WARNING_STOP )
      { S7_GenerateENO := "TRUE" } Move(in := 2, out1 => "DB7238_HMI_WINCC_OVERVIEW".U02_STA3_ALARMS_LED_STATUS)
   END_RUNG
   RUNG wire#w1
      I_Contact( "DB440_MACHINE_ALARM_DECODING".ALARMS_UNIT_02.ST3_CLADDING.ALARM )
      Contact( "DB440_MACHINE_ALARM_DECODING".ALARMS_UNIT_02.ST3_CLADDING.WARNING_STOP )
      { S7_GenerateENO := "TRUE" } Move(in := 1, out1 => "DB7238_HMI_WINCC_OVERVIEW".U02_STA3_ALARMS_LED_STATUS)
   END_RUNG
   RUNG wire#w1
      Contact( "DB440_MACHINE_ALARM_DECODING".ALARMS_UNIT_02.ST3_CLADDING.ALARM )
      { S7_GenerateENO := "TRUE" } Move(in := 0, out1 => "DB7238_HMI_WINCC_OVERVIEW".U02_STA3_ALARMS_LED_STATUS)
   END_RUNG
   // the same network as SCL:
   IF "M_ONE" AND NOT "DB440_MACHINE_ALARM_DECODING".ALARMS_UNIT_02.ST3_CLADDING.ALARM AND NOT "DB440_MACHINE_ALARM_DECODING".ALARMS_UNIT_02.ST3_CLADDING.WARNING_STOP THEN
       "DB7238_HMI_WINCC_OVERVIEW".U02_STA3_ALARMS_LED_STATUS := 2;
   END_IF;
   IF "M_ONE" AND NOT "DB440_MACHINE_ALARM_DECODING".ALARMS_UNIT_02.ST3_CLADDING.ALARM AND "DB440_MACHINE_ALARM_DECODING".ALARMS_UNIT_02.ST3_CLADDING.WARNING_STOP THEN
       "DB7238_HMI_WINCC_OVERVIEW".U02_STA3_ALARMS_LED_STATUS := 1;
   END_IF;
   IF "M_ONE" AND "DB440_MACHINE_ALARM_DECODING".ALARMS_UNIT_02.ST3_CLADDING.ALARM THEN
       "DB7238_HMI_WINCC_OVERVIEW".U02_STA3_ALARMS_LED_STATUS := 0;
   END_IF;
END_REGION

REGION Network 35: UNIT 02 STATION 4 ALARMS AND WARNINGS LED STATUS
   RUNG wire#powerrail
      Contact( "M_ONE" )
      wire#w1
      I_Contact( "DB440_MACHINE_ALARM_DECODING".ALARMS_UNIT_02.ST4_CLEANING.ALARM )
      I_Contact( "DB440_MACHINE_ALARM_DECODING".ALARMS_UNIT_02.ST4_CLEANING.WARNING_STOP )
      { S7_GenerateENO := "TRUE" } Move(in := 2, out1 => "DB7238_HMI_WINCC_OVERVIEW".U02_STA4_ALARMS_LED_STATUS)
   END_RUNG
   RUNG wire#w1
      I_Contact( "DB440_MACHINE_ALARM_DECODING".ALARMS_UNIT_02.ST4_CLEANING.ALARM )
      Contact( "DB440_MACHINE_ALARM_DECODING".ALARMS_UNIT_02.ST4_CLEANING.WARNING_STOP )
      { S7_GenerateENO := "TRUE" } Move(in := 1, out1 => "DB7238_HMI_WINCC_OVERVIEW".U02_STA4_ALARMS_LED_STATUS)
   END_RUNG
   RUNG wire#w1
      Contact( "DB440_MACHINE_ALARM_DECODING".ALARMS_UNIT_02.ST4_CLEANING.ALARM )
      { S7_GenerateENO := "TRUE" } Move(in := 0, out1 => "DB7238_HMI_WINCC_OVERVIEW".U02_STA4_ALARMS_LED_STATUS)
   END_RUNG
   // the same network as SCL:
   IF "M_ONE" AND NOT "DB440_MACHINE_ALARM_DECODING".ALARMS_UNIT_02.ST4_CLEANING.ALARM AND NOT "DB440_MACHINE_ALARM_DECODING".ALARMS_UNIT_02.ST4_CLEANING.WARNING_STOP THEN
       "DB7238_HMI_WINCC_OVERVIEW".U02_STA4_ALARMS_LED_STATUS := 2;
   END_IF;
   IF "M_ONE" AND NOT "DB440_MACHINE_ALARM_DECODING".ALARMS_UNIT_02.ST4_CLEANING.ALARM AND "DB440_MACHINE_ALARM_DECODING".ALARMS_UNIT_02.ST4_CLEANING.WARNING_STOP THEN
       "DB7238_HMI_WINCC_OVERVIEW".U02_STA4_ALARMS_LED_STATUS := 1;
   END_IF;
   IF "M_ONE" AND "DB440_MACHINE_ALARM_DECODING".ALARMS_UNIT_02.ST4_CLEANING.ALARM THEN
       "DB7238_HMI_WINCC_OVERVIEW".U02_STA4_ALARMS_LED_STATUS := 0;
   END_IF;
END_REGION

REGION Network 36: UNIT 02 ALL FIXTURES CLAMP ALARMS
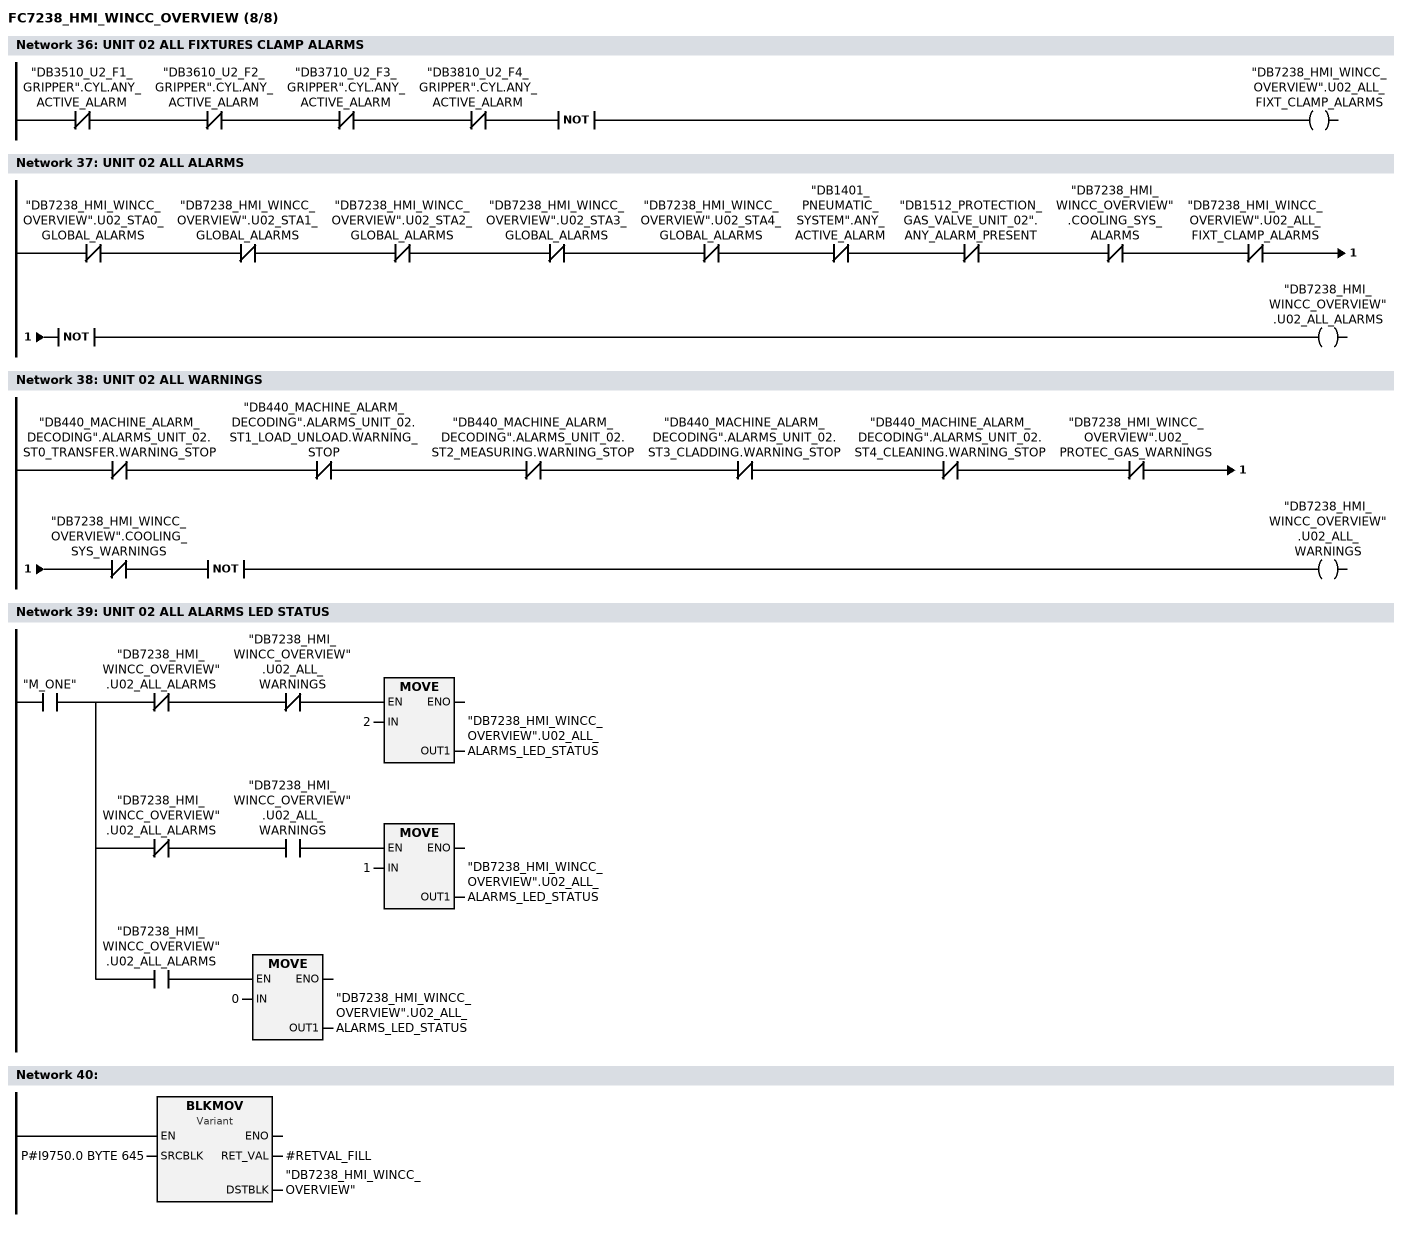
   RUNG wire#powerrail
      I_Contact( "DB3510_U2_F1_GRIPPER".CYL.ANY_ACTIVE_ALARM )
      I_Contact( "DB3610_U2_F2_GRIPPER".CYL.ANY_ACTIVE_ALARM )
      I_Contact( "DB3710_U2_F3_GRIPPER".CYL.ANY_ACTIVE_ALARM )
      I_Contact( "DB3810_U2_F4_GRIPPER".CYL.ANY_ACTIVE_ALARM )
      Not()
      Coil( "DB7238_HMI_WINCC_OVERVIEW".U02_ALL_FIXT_CLAMP_ALARMS )
   END_RUNG
   // the same network as SCL:
   "DB7238_HMI_WINCC_OVERVIEW".U02_ALL_FIXT_CLAMP_ALARMS := NOT (NOT "DB3510_U2_F1_GRIPPER".CYL.ANY_ACTIVE_ALARM AND NOT "DB3610_U2_F2_GRIPPER".CYL.ANY_ACTIVE_ALARM AND NOT "DB3710_U2_F3_GRIPPER".CYL.ANY_ACTIVE_ALARM AND NOT "DB3810_U2_F4_GRIPPER".CYL.ANY_ACTIVE_ALARM);
END_REGION

REGION Network 37: UNIT 02 ALL ALARMS
   RUNG wire#powerrail
      I_Contact( "DB7238_HMI_WINCC_OVERVIEW".U02_STA0_GLOBAL_ALARMS )
      I_Contact( "DB7238_HMI_WINCC_OVERVIEW".U02_STA1_GLOBAL_ALARMS )
      I_Contact( "DB7238_HMI_WINCC_OVERVIEW".U02_STA2_GLOBAL_ALARMS )
      I_Contact( "DB7238_HMI_WINCC_OVERVIEW".U02_STA3_GLOBAL_ALARMS )
      I_Contact( "DB7238_HMI_WINCC_OVERVIEW".U02_STA4_GLOBAL_ALARMS )
      I_Contact( "DB1401_PNEUMATIC_SYSTEM".ANY_ACTIVE_ALARM )
      I_Contact( "DB1512_PROTECTION_GAS_VALVE_UNIT_02".ANY_ALARM_PRESENT )
      I_Contact( "DB7238_HMI_WINCC_OVERVIEW".COOLING_SYS_ALARMS )
      I_Contact( "DB7238_HMI_WINCC_OVERVIEW".U02_ALL_FIXT_CLAMP_ALARMS )
      Not()
      Coil( "DB7238_HMI_WINCC_OVERVIEW".U02_ALL_ALARMS )
   END_RUNG
   // the same network as SCL:
   "DB7238_HMI_WINCC_OVERVIEW".U02_ALL_ALARMS := NOT (NOT "DB7238_HMI_WINCC_OVERVIEW".U02_STA0_GLOBAL_ALARMS AND NOT "DB7238_HMI_WINCC_OVERVIEW".U02_STA1_GLOBAL_ALARMS AND NOT "DB7238_HMI_WINCC_OVERVIEW".U02_STA2_GLOBAL_ALARMS AND NOT "DB7238_HMI_WINCC_OVERVIEW".U02_STA3_GLOBAL_ALARMS AND NOT "DB7238_HMI_WINCC_OVERVIEW".U02_STA4_GLOBAL_ALARMS AND NOT "DB1401_PNEUMATIC_SYSTEM".ANY_ACTIVE_ALARM AND NOT "DB1512_PROTECTION_GAS_VALVE_UNIT_02".ANY_ALARM_PRESENT AND NOT "DB7238_HMI_WINCC_OVERVIEW".COOLING_SYS_ALARMS AND NOT "DB7238_HMI_WINCC_OVERVIEW".U02_ALL_FIXT_CLAMP_ALARMS);
END_REGION

REGION Network 38: UNIT 02 ALL WARNINGS
   RUNG wire#powerrail
      I_Contact( "DB440_MACHINE_ALARM_DECODING".ALARMS_UNIT_02.ST0_TRANSFER.WARNING_STOP )
      I_Contact( "DB440_MACHINE_ALARM_DECODING".ALARMS_UNIT_02.ST1_LOAD_UNLOAD.WARNING_STOP )
      I_Contact( "DB440_MACHINE_ALARM_DECODING".ALARMS_UNIT_02.ST2_MEASURING.WARNING_STOP )
      I_Contact( "DB440_MACHINE_ALARM_DECODING".ALARMS_UNIT_02.ST3_CLADDING.WARNING_STOP )
      I_Contact( "DB440_MACHINE_ALARM_DECODING".ALARMS_UNIT_02.ST4_CLEANING.WARNING_STOP )
      I_Contact( "DB7238_HMI_WINCC_OVERVIEW".U02_PROTEC_GAS_WARNINGS )
      I_Contact( "DB7238_HMI_WINCC_OVERVIEW".COOLING_SYS_WARNINGS )
      Not()
      Coil( "DB7238_HMI_WINCC_OVERVIEW".U02_ALL_WARNINGS )
   END_RUNG
   // the same network as SCL:
   "DB7238_HMI_WINCC_OVERVIEW".U02_ALL_WARNINGS := NOT (NOT "DB440_MACHINE_ALARM_DECODING".ALARMS_UNIT_02.ST0_TRANSFER.WARNING_STOP AND NOT "DB440_MACHINE_ALARM_DECODING".ALARMS_UNIT_02.ST1_LOAD_UNLOAD.WARNING_STOP AND NOT "DB440_MACHINE_ALARM_DECODING".ALARMS_UNIT_02.ST2_MEASURING.WARNING_STOP AND NOT "DB440_MACHINE_ALARM_DECODING".ALARMS_UNIT_02.ST3_CLADDING.WARNING_STOP AND NOT "DB440_MACHINE_ALARM_DECODING".ALARMS_UNIT_02.ST4_CLEANING.WARNING_STOP AND NOT "DB7238_HMI_WINCC_OVERVIEW".U02_PROTEC_GAS_WARNINGS AND NOT "DB7238_HMI_WINCC_OVERVIEW".COOLING_SYS_WARNINGS);
END_REGION

REGION Network 39: UNIT 02 ALL ALARMS LED STATUS
   RUNG wire#powerrail
      Contact( "M_ONE" )
      wire#w1
      I_Contact( "DB7238_HMI_WINCC_OVERVIEW".U02_ALL_ALARMS )
      I_Contact( "DB7238_HMI_WINCC_OVERVIEW".U02_ALL_WARNINGS )
      { S7_GenerateENO := "TRUE" } Move(in := 2, out1 => "DB7238_HMI_WINCC_OVERVIEW".U02_ALL_ALARMS_LED_STATUS)
   END_RUNG
   RUNG wire#w1
      I_Contact( "DB7238_HMI_WINCC_OVERVIEW".U02_ALL_ALARMS )
      Contact( "DB7238_HMI_WINCC_OVERVIEW".U02_ALL_WARNINGS )
      { S7_GenerateENO := "TRUE" } Move(in := 1, out1 => "DB7238_HMI_WINCC_OVERVIEW".U02_ALL_ALARMS_LED_STATUS)
   END_RUNG
   RUNG wire#w1
      Contact( "DB7238_HMI_WINCC_OVERVIEW".U02_ALL_ALARMS )
      { S7_GenerateENO := "TRUE" } Move(in := 0, out1 => "DB7238_HMI_WINCC_OVERVIEW".U02_ALL_ALARMS_LED_STATUS)
   END_RUNG
   // the same network as SCL:
   IF "M_ONE" AND NOT "DB7238_HMI_WINCC_OVERVIEW".U02_ALL_ALARMS AND NOT "DB7238_HMI_WINCC_OVERVIEW".U02_ALL_WARNINGS THEN
       "DB7238_HMI_WINCC_OVERVIEW".U02_ALL_ALARMS_LED_STATUS := 2;
   END_IF;
   IF "M_ONE" AND NOT "DB7238_HMI_WINCC_OVERVIEW".U02_ALL_ALARMS AND "DB7238_HMI_WINCC_OVERVIEW".U02_ALL_WARNINGS THEN
       "DB7238_HMI_WINCC_OVERVIEW".U02_ALL_ALARMS_LED_STATUS := 1;
   END_IF;
   IF "M_ONE" AND "DB7238_HMI_WINCC_OVERVIEW".U02_ALL_ALARMS THEN
       "DB7238_HMI_WINCC_OVERVIEW".U02_ALL_ALARMS_LED_STATUS := 0;
   END_IF;
END_REGION

REGION Network 40
   RUNG wire#powerrail
      { S7_Templates := "blk_type := Variant" } BLKMOV(SRCBLK := P#I9750.0 BYTE 645, RET_VAL => #RETVAL_FILL, DSTBLK => "DB7238_HMI_WINCC_OVERVIEW")
   END_RUNG
   // the same network as SCL:
   #RETVAL_FILL := BLKMOV(SRCBLK := P#I9750.0 BYTE 645, DSTBLK => "DB7238_HMI_WINCC_OVERVIEW");
END_REGION
END_FUNCTION
